// Check duration for each phase
positionExtrema := ruckig._profiles[0].Bound();
AssertEquals_LREAL(0.13645534129957551106, positionExtrema.Tmax, 1E-9, message:='Profile[0] Tmax incorrect');
AssertEquals_LREAL(-9.75706058924097519025, positionExtrema.Maximum, 1E-9, message:='Profile[0] maximum incorrect');
AssertEquals_LREAL(0.18561602058648316027, positionExtrema.Tmin, 1E-9, message:='Profile[0] Tmin incorrect');
AssertEquals_LREAL(-27.59745181479642894828, positionExtrema.Minimum, 1E-9, message:='Profile[0] minimum incorrect');

positionExtrema := ruckig._profiles[1].Bound();
AssertEquals_LREAL(0.18561602058648316027, positionExtrema.Tmax, 1E-9, message:='Profile[1] Tmax incorrect');
AssertEquals_LREAL(97.62295145618037395252, positionExtrema.Maximum, 1E-9, message:='Profile[1] maximum incorrect');
AssertEquals_LREAL(0.07177100934221260220, positionExtrema.Tmin, 1E-9, message:='Profile[1] Tmin incorrect');
AssertEquals_LREAL(33.68002966797480723926, positionExtrema.Minimum, 1E-9, message:='Profile[1] minimum incorrect');

positionExtrema := ruckig._profiles[2].Bound();
AssertEquals_LREAL(0.17125230195322679871, positionExtrema.Tmax, 1E-9, message:='Profile[2] Tmax incorrect');
AssertEquals_LREAL(-3.71520543795192104142, positionExtrema.Maximum, 1E-9, message:='Profile[2] maximum incorrect');
AssertEquals_LREAL(0.02823480242135182477, positionExtrema.Tmin, 1E-9, message:='Profile[2] Tmin incorrect');
AssertEquals_LREAL(-58.80508937654931855832, positionExtrema.Minimum, 1E-9, message:='Profile[2] minimum incorrect');
   

TEST_FINISHED();
END_METHOD

METHOD Test_Trajectory_HasTargetVelocity_17
VAR_INST
  ruckig : Struckig.Otg(0.001, 3) := (
  
    Synchronization := SynchronizationType.TimeSync,        
    MaxVelocity := [ 2000.00000000000000000000, 2000.00000000000000000000, 2000.00000000000000000000 ],
    MaxAcceleration := [ 20000.00000000000000000000, 20000.00000000000000000000, 20000.00000000000000000000 ],
    MaxJerk := [ 800000.00000000000000000000, 800000.00000000000000000000, 800000.00000000000000000000 ],
    CurrentPosition := [ 29.09201686409977583025, 26.79555889099025023370, -2.56405583533239678218 ],
    CurrentVelocity := [ -865.74515531652343725000, -446.66804096341445529106, 715.70430296883705523214 ],
    CurrentAcceleration := [ -419.53152796798531198874, 3725.90159379652868665289, 3083.71115629947962588631 ],
    TargetPosition := [ -5.98395477362167582669, 85.98880639059657937651, -77.56683653164213865239 ],
    TargetVelocity := [ -487.77111778150026566436, 597.93719815311010279402, -19.66112295679818089411 ],
    TargetAcceleration := [ 0.00000000000000000000, 0.00000000000000000000, 0.00000000000000000000 ]
  );
  
  positionExtrema : Struckig.ProfileBound;
END_VAR
TEST('Trajectory_HasTargetVelocity_17');

ruckig();

// Check total duration of profiles
AssertEquals_LREAL(Expected := 0.20727577661691312660, Actual := ruckig.Duration, DELTA := 1E-8, Message := 'Duration incorrect');

// Check duration for each phase
positionExtrema := ruckig._profiles[0].Bound();
AssertEquals_LREAL(0.00000000000000000000, positionExtrema.Tmax, 1E-9, message:='Profile[0] Tmax incorrect');
AssertEquals_LREAL(29.09201686409977583025, positionExtrema.Maximum, 1E-9, message:='Profile[0] maximum incorrect');
AssertEquals_LREAL(0.20727577661691309885, positionExtrema.Tmin, 1E-9, message:='Profile[0] Tmin incorrect');
AssertEquals_LREAL(-5.98395477362167582669, positionExtrema.Minimum, 1E-9, message:='Profile[0] minimum incorrect');

positionExtrema := ruckig._profiles[1].Bound();
AssertEquals_LREAL(0.20727577661691312660, positionExtrema.Tmax, 1E-9, message:='Profile[1] Tmax incorrect');
AssertEquals_LREAL(85.98880639059657937651, positionExtrema.Maximum, 1E-9, message:='Profile[1] maximum incorrect');
AssertEquals_LREAL(0.03742622748756373185, positionExtrema.Tmin, 1E-9, message:='Profile[1] Tmin incorrect');
AssertEquals_LREAL(19.01299187494276665689, positionExtrema.Minimum, 1E-9, message:='Profile[1] minimum incorrect');

positionExtrema := ruckig._profiles[2].Bound();
AssertEquals_LREAL(0.02885463894537435015, positionExtrema.Tmax, 1E-9, message:='Profile[2] Tmax incorrect');
AssertEquals_LREAL(16.16785534073141050726, positionExtrema.Maximum, 1E-9, message:='Profile[2] maximum incorrect');
AssertEquals_LREAL(0.20727577661691312660, positionExtrema.Tmin, 1E-9, message:='Profile[2] Tmin incorrect');
AssertEquals_LREAL(-77.56683653164213865239, positionExtrema.Minimum, 1E-9, message:='Profile[2] minimum incorrect');
   

TEST_FINISHED();
END_METHOD

METHOD Test_Trajectory_HasTargetVelocity_19
VAR_INST
  ruckig : Struckig.Otg(0.001, 3) := (
  
    Synchronization := SynchronizationType.TimeSync,        
    MaxVelocity := [ 2000.00000000000000000000, 2000.00000000000000000000, 2000.00000000000000000000 ],
    MaxAcceleration := [ 20000.00000000000000000000, 20000.00000000000000000000, 20000.00000000000000000000 ],
    MaxJerk := [ 800000.00000000000000000000, 800000.00000000000000000000, 800000.00000000000000000000 ],
    CurrentPosition := [ 80.71252725401120642346, 44.88025621959243949277, -12.15149697459605704353 ],
    CurrentVelocity := [ -948.15980924147334008012, -489.88340864146471176355, -827.37383618723242761916 ],
    CurrentAcceleration := [ -3514.54219608491530379979, -6906.59296787188577582128, 1315.32694212922615406569 ],
    TargetPosition := [ 59.95790772621657538366, -72.33902659712904892331, -15.83444921441858355138 ],
    TargetVelocity := [ -459.58488479420384464902, 187.24245841899073639070, 921.25657886294084164547 ],
    TargetAcceleration := [ 0.00000000000000000000, 0.00000000000000000000, 0.00000000000000000000 ]
  );
  
  positionExtrema : Struckig.ProfileBound;
END_VAR
TEST('Trajectory_HasTargetVelocity_19');

ruckig();

// Check total duration of profiles
AssertEquals_LREAL(Expected := 0.18063360611716061666, Actual := ruckig.Duration, DELTA := 1E-8, Message := 'Duration incorrect');

// Check duration for each phase
positionExtrema := ruckig._profiles[0].Bound();
AssertEquals_LREAL(0.00000000000000000000, positionExtrema.Tmax, 1E-9, message:='Profile[0] Tmax incorrect');
AssertEquals_LREAL(80.71252725401120642346, positionExtrema.Maximum, 1E-9, message:='Profile[0] maximum incorrect');
AssertEquals_LREAL(0.07992076514931607811, positionExtrema.Tmin, 1E-9, message:='Profile[0] Tmin incorrect');
AssertEquals_LREAL(44.57478735687137572086, positionExtrema.Minimum, 1E-9, message:='Profile[0] minimum incorrect');

positionExtrema := ruckig._profiles[1].Bound();
AssertEquals_LREAL(0.00000000000000000000, positionExtrema.Tmax, 1E-9, message:='Profile[1] Tmax incorrect');
AssertEquals_LREAL(44.88025621959243949277, positionExtrema.Maximum, 1E-9, message:='Profile[1] maximum incorrect');
AssertEquals_LREAL(0.15899784530207772271, positionExtrema.Tmin, 1E-9, message:='Profile[1] Tmin incorrect');
AssertEquals_LREAL(-75.03978196031663117083, positionExtrema.Minimum, 1E-9, message:='Profile[1] minimum incorrect');

positionExtrema := ruckig._profiles[2].Bound();
AssertEquals_LREAL(0.00000000000000000000, positionExtrema.Tmax, 1E-9, message:='Profile[2] Tmax incorrect');
AssertEquals_LREAL(-12.15149697459605704353, positionExtrema.Maximum, 1E-9, message:='Profile[2] maximum incorrect');
AssertEquals_LREAL(0.12139203206320470230, positionExtrema.Tmin, 1E-9, message:='Profile[2] Tmin incorrect');
AssertEquals_LREAL(-48.06891878044748267484, positionExtrema.Minimum, 1E-9, message:='Profile[2] minimum incorrect');
   

TEST_FINISHED();
END_METHOD

METHOD Test_Trajectory_HasTargetVelocity_20
VAR_INST
  ruckig : Struckig.Otg(0.001, 3) := (
  
    Synchronization := SynchronizationType.TimeSync,        
    MaxVelocity := [ 2000.00000000000000000000, 2000.00000000000000000000, 2000.00000000000000000000 ],
    MaxAcceleration := [ 20000.00000000000000000000, 20000.00000000000000000000, 20000.00000000000000000000 ],
    MaxJerk := [ 800000.00000000000000000000, 800000.00000000000000000000, 800000.00000000000000000000 ],
    CurrentPosition := [ 83.23209059023531608545, -91.01412900146218021291, -45.02313424428616883688 ],
    CurrentVelocity := [ 478.85135262944709211297, 941.48041828651457763044, 233.77464784894095828349 ],
    CurrentAcceleration := [ 4901.95944988452902180143, -711.94018044516997179016, -6268.14311607610761711840 ],
    TargetPosition := [ -60.31306848800090847362, -76.05388552166272120303, -77.88363097381802901964 ],
    TargetVelocity := [ -28.42585943091080480372, 112.61218905881105456501, -518.94659889602689872845 ],
    TargetAcceleration := [ 0.00000000000000000000, 0.00000000000000000000, 0.00000000000000000000 ]
  );
  
  positionExtrema : Struckig.ProfileBound;
END_VAR
TEST('Trajectory_HasTargetVelocity_20');

ruckig();

// Check total duration of profiles
AssertEquals_LREAL(Expected := 0.23417815197351798950, Actual := ruckig.Duration, DELTA := 1E-8, Message := 'Duration incorrect');

// Check duration for each phase
positionExtrema := ruckig._profiles[0].Bound();
AssertEquals_LREAL(0.03112744931235566018, positionExtrema.Tmax, 1E-9, message:='Profile[0] Tmax incorrect');
AssertEquals_LREAL(96.49098387500299622843, positionExtrema.Maximum, 1E-9, message:='Profile[0] maximum incorrect');
AssertEquals_LREAL(0.23417815197351798950, positionExtrema.Tmin, 1E-9, message:='Profile[0] Tmin incorrect');
AssertEquals_LREAL(-60.31306848800090847362, positionExtrema.Minimum, 1E-9, message:='Profile[0] minimum incorrect');

positionExtrema := ruckig._profiles[1].Bound();
AssertEquals_LREAL(0.05967434054652072384, positionExtrema.Tmax, 1E-9, message:='Profile[1] Tmax incorrect');
AssertEquals_LREAL(-58.39013538569540884282, positionExtrema.Maximum, 1E-9, message:='Profile[1] maximum incorrect');
AssertEquals_LREAL(0.00000000000000000000, positionExtrema.Tmin, 1E-9, message:='Profile[1] Tmin incorrect');
AssertEquals_LREAL(-91.01412900146218021291, positionExtrema.Minimum, 1E-9, message:='Profile[1] minimum incorrect');

positionExtrema := ruckig._profiles[2].Bound();
AssertEquals_LREAL(0.01824400060866057660, positionExtrema.Tmax, 1E-9, message:='Profile[2] Tmax incorrect');
AssertEquals_LREAL(-42.59202121085846926007, positionExtrema.Maximum, 1E-9, message:='Profile[2] maximum incorrect');
AssertEquals_LREAL(0.23417815197351793399, positionExtrema.Tmin, 1E-9, message:='Profile[2] Tmin incorrect');
AssertEquals_LREAL(-77.88363097381802901964, positionExtrema.Minimum, 1E-9, message:='Profile[2] minimum incorrect');
   

TEST_FINISHED();
END_METHOD

METHOD Test_Trajectory_HasTargetVelocity_21
VAR_INST
  ruckig : Struckig.Otg(0.001, 3) := (
  
    Synchronization := SynchronizationType.TimeSync,        
    MaxVelocity := [ 2000.00000000000000000000, 2000.00000000000000000000, 2000.00000000000000000000 ],
    MaxAcceleration := [ 20000.00000000000000000000, 20000.00000000000000000000, 20000.00000000000000000000 ],
    MaxJerk := [ 800000.00000000000000000000, 800000.00000000000000000000, 800000.00000000000000000000 ],
    CurrentPosition := [ -90.18105588355366819542, 11.40426253106177512109, -96.96426550769332664004 ],
    CurrentVelocity := [ 268.68366267133455949079, -230.39092451139003969729, 217.37624370386924965715 ],
    CurrentAcceleration := [ 6950.36478944877671892755, -1973.79956680386658263160, 9973.29839097329022479244 ],
    TargetPosition := [ 56.23264204687242795444, 89.78670651839811966965, 35.61941562712866016227 ],
    TargetVelocity := [ -748.79294734560005508683, 279.58550802373474652995, 329.97469268802092301485 ],
    TargetAcceleration := [ 0.00000000000000000000, 0.00000000000000000000, 0.00000000000000000000 ]
  );
  
  positionExtrema : Struckig.ProfileBound;
END_VAR
TEST('Trajectory_HasTargetVelocity_21');

ruckig();

// Check total duration of profiles
AssertEquals_LREAL(Expected := 0.22811513995984869507, Actual := ruckig.Duration, DELTA := 1E-8, Message := 'Duration incorrect');

// Check duration for each phase
positionExtrema := ruckig._profiles[0].Bound();
AssertEquals_LREAL(0.20311513995984870062, positionExtrema.Tmax, 1E-9, message:='Profile[0] Tmax incorrect');
AssertEquals_LREAL(72.86913239717907231352, positionExtrema.Maximum, 1E-9, message:='Profile[0] maximum incorrect');
AssertEquals_LREAL(0.00000000000000000000, positionExtrema.Tmin, 1E-9, message:='Profile[0] Tmin incorrect');
AssertEquals_LREAL(-90.18105588355366819542, positionExtrema.Minimum, 1E-9, message:='Profile[0] minimum incorrect');

positionExtrema := ruckig._profiles[1].Bound();
AssertEquals_LREAL(0.22811513995984869507, positionExtrema.Tmax, 1E-9, message:='Profile[1] Tmax incorrect');
AssertEquals_LREAL(89.78670651839811966965, positionExtrema.Maximum, 1E-9, message:='Profile[1] maximum incorrect');
AssertEquals_LREAL(0.02659326510902134191, positionExtrema.Tmin, 1E-9, message:='Profile[1] Tmin incorrect');
AssertEquals_LREAL(7.08705215721043568777, positionExtrema.Minimum, 1E-9, message:='Profile[1] minimum incorrect');

positionExtrema := ruckig._profiles[2].Bound();
AssertEquals_LREAL(0.22811513995984869507, positionExtrema.Tmax, 1E-9, message:='Profile[2] Tmax incorrect');
AssertEquals_LREAL(35.61941562712866016227, positionExtrema.Maximum, 1E-9, message:='Profile[2] maximum incorrect');
AssertEquals_LREAL(0.00000000000000000000, positionExtrema.Tmin, 1E-9, message:='Profile[2] Tmin incorrect');
AssertEquals_LREAL(-96.96426550769332664004, positionExtrema.Minimum, 1E-9, message:='Profile[2] minimum incorrect');
   

TEST_FINISHED();
END_METHOD

METHOD Test_Trajectory_HasTargetVelocity_22
VAR_INST
  ruckig : Struckig.Otg(0.001, 3) := (
  
    Synchronization := SynchronizationType.TimeSync,        
    MaxVelocity := [ 2000.00000000000000000000, 2000.00000000000000000000, 2000.00000000000000000000 ],
    MaxAcceleration := [ 20000.00000000000000000000, 20000.00000000000000000000, 20000.00000000000000000000 ],
    MaxJerk := [ 800000.00000000000000000000, 800000.00000000000000000000, 800000.00000000000000000000 ],
    CurrentPosition := [ -67.41063214653675572663, -34.84504669460216064181, 71.90844709145784463544 ],
    CurrentVelocity := [ -627.45307756820307076850, -697.56722522760969695810, -660.83791164052786371030 ],
    CurrentAcceleration := [ -7277.38846981411006709095, -2750.24172428648398636142, -978.85332476885741925798 ],
    TargetPosition := [ -57.66574268409263481772, -88.27667420321476754452, 96.97655926730644182499 ],
    TargetVelocity := [ -610.75498065854083051818, -654.20857948874163412256, 336.03100506981877515500 ],
    TargetAcceleration := [ 0.00000000000000000000, 0.00000000000000000000, 0.00000000000000000000 ]
  );
  
  positionExtrema : Struckig.ProfileBound;
END_VAR
TEST('Trajectory_HasTargetVelocity_22');

ruckig();

// Check total duration of profiles
AssertEquals_LREAL(Expected := 0.20245104517991782678, Actual := ruckig.Duration, DELTA := 1E-8, Message := 'Duration incorrect');

// Check duration for each phase
positionExtrema := ruckig._profiles[0].Bound();
AssertEquals_LREAL(0.17745104517991783233, positionExtrema.Tmax, 1E-9, message:='Profile[0] Tmax incorrect');
AssertEquals_LREAL(-44.48020150096243696680, positionExtrema.Maximum, 1E-9, message:='Profile[0] maximum incorrect');
AssertEquals_LREAL(0.03409673558726764031, positionExtrema.Tmin, 1E-9, message:='Profile[0] Tmin incorrect');
AssertEquals_LREAL(-87.74964255933160472978, positionExtrema.Minimum, 1E-9, message:='Profile[0] minimum incorrect');

positionExtrema := ruckig._profiles[1].Bound();
AssertEquals_LREAL(0.00000000000000000000, positionExtrema.Tmax, 1E-9, message:='Profile[1] Tmax incorrect');
AssertEquals_LREAL(-34.84504669460216064181, positionExtrema.Maximum, 1E-9, message:='Profile[1] maximum incorrect');
AssertEquals_LREAL(0.20245104517991779902, positionExtrema.Tmin, 1E-9, message:='Profile[1] Tmin incorrect');
AssertEquals_LREAL(-88.27667420321476754452, positionExtrema.Minimum, 1E-9, message:='Profile[1] minimum incorrect');

positionExtrema := ruckig._profiles[2].Bound();
AssertEquals_LREAL(0.20245104517991782678, positionExtrema.Tmax, 1E-9, message:='Profile[2] Tmax incorrect');
AssertEquals_LREAL(96.97655926730644182499, positionExtrema.Maximum, 1E-9, message:='Profile[2] maximum incorrect');
AssertEquals_LREAL(0.04944613992821229875, positionExtrema.Tmin, 1E-9, message:='Profile[2] Tmin incorrect');
AssertEquals_LREAL(52.48505260032155916861, positionExtrema.Minimum, 1E-9, message:='Profile[2] minimum incorrect');
   

TEST_FINISHED();
END_METHOD

METHOD Test_Trajectory_HasTargetVelocity_27
VAR_INST
  ruckig : Struckig.Otg(0.001, 3) := (
  
    Synchronization := SynchronizationType.TimeSync,        
    MaxVelocity := [ 2000.00000000000000000000, 2000.00000000000000000000, 2000.00000000000000000000 ],
    MaxAcceleration := [ 20000.00000000000000000000, 20000.00000000000000000000, 20000.00000000000000000000 ],
    MaxJerk := [ 800000.00000000000000000000, 800000.00000000000000000000, 800000.00000000000000000000 ],
    CurrentPosition := [ -29.47354331486815226526, 27.93495185982479256381, 25.04726746624395161689 ],
    CurrentVelocity := [ -230.41514646826715306815, -990.61050993041703804920, -730.89168845843755661917 ],
    CurrentAcceleration := [ 8742.55847153794820769690, 5915.09847409233043435961, 4511.30118221045631798916 ],
    TargetPosition := [ -46.00476070479609091990, -93.63874889974350423927, -84.98442462304464584122 ],
    TargetVelocity := [ 6.00636834947817987995, -353.84810777792165481515, -981.55918901141831156565 ],
    TargetAcceleration := [ 0.00000000000000000000, 0.00000000000000000000, 0.00000000000000000000 ]
  );
  
  positionExtrema : Struckig.ProfileBound;
END_VAR
TEST('Trajectory_HasTargetVelocity_27');

ruckig();

// Check total duration of profiles
AssertEquals_LREAL(Expected := 0.12586715797260131233, Actual := ruckig.Duration, DELTA := 1E-8, Message := 'Duration incorrect');

// Check duration for each phase
positionExtrema := ruckig._profiles[0].Bound();
AssertEquals_LREAL(0.00000000000000000000, positionExtrema.Tmax, 1E-9, message:='Profile[0] Tmax incorrect');
AssertEquals_LREAL(-29.47354331486815226526, positionExtrema.Maximum, 1E-9, message:='Profile[0] maximum incorrect');
AssertEquals_LREAL(0.12199211979553833962, positionExtrema.Tmin, 1E-9, message:='Profile[0] Tmin incorrect');
AssertEquals_LREAL(-46.02027730923590809198, positionExtrema.Minimum, 1E-9, message:='Profile[0] minimum incorrect');

positionExtrema := ruckig._profiles[1].Bound();
AssertEquals_LREAL(0.00000000000000000000, positionExtrema.Tmax, 1E-9, message:='Profile[1] Tmax incorrect');
AssertEquals_LREAL(27.93495185982479256381, positionExtrema.Maximum, 1E-9, message:='Profile[1] maximum incorrect');
AssertEquals_LREAL(0.12586715797260131233, positionExtrema.Tmin, 1E-9, message:='Profile[1] Tmin incorrect');
AssertEquals_LREAL(-93.63874889974350423927, positionExtrema.Minimum, 1E-9, message:='Profile[1] minimum incorrect');

positionExtrema := ruckig._profiles[2].Bound();
AssertEquals_LREAL(0.00000000000000000000, positionExtrema.Tmax, 1E-9, message:='Profile[2] Tmax incorrect');
AssertEquals_LREAL(25.04726746624395161689, positionExtrema.Maximum, 1E-9, message:='Profile[2] maximum incorrect');
AssertEquals_LREAL(0.12586715797260131233, positionExtrema.Tmin, 1E-9, message:='Profile[2] Tmin incorrect');
AssertEquals_LREAL(-84.98442462304464584122, positionExtrema.Minimum, 1E-9, message:='Profile[2] minimum incorrect');
   

TEST_FINISHED();
END_METHOD

METHOD Test_Trajectory_HasTargetVelocity_3
VAR_INST
  ruckig : Struckig.Otg(0.001, 3) := (
  
    Synchronization := SynchronizationType.TimeSync,        
    MaxVelocity := [ 2000.00000000000000000000, 2000.00000000000000000000, 2000.00000000000000000000 ],
    MaxAcceleration := [ 20000.00000000000000000000, 20000.00000000000000000000, 20000.00000000000000000000 ],
    MaxJerk := [ 800000.00000000000000000000, 800000.00000000000000000000, 800000.00000000000000000000 ],
    CurrentPosition := [ 26.53957997779905042535, -93.07095602825359037524, -22.16503543192527558858 ],
    CurrentVelocity := [ -978.47395774087203790259, 118.42434690487039006257, -240.97450183146906965703 ],
    CurrentAcceleration := [ 6077.24253675401814689394, 6138.16243012785889732186, -287.73427625073964009061 ],
    TargetPosition := [ -74.88074053142992170251, -34.02780494232007413302, 79.44667149152985530236 ],
    TargetVelocity := [ 90.05732775263027178880, 511.77846374302612275642, 384.28752753365688477061 ],
    TargetAcceleration := [ 0.00000000000000000000, 0.00000000000000000000, 0.00000000000000000000 ]
  );
  
  positionExtrema : Struckig.ProfileBound;
END_VAR
TEST('Trajectory_HasTargetVelocity_3');

ruckig();

// Check total duration of profiles
AssertEquals_LREAL(Expected := 0.16528629612631601242, Actual := ruckig.Duration, DELTA := 1E-8, Message := 'Duration incorrect');

// Check duration for each phase
positionExtrema := ruckig._profiles[0].Bound();
AssertEquals_LREAL(0.00000000000000000000, positionExtrema.Tmax, 1E-9, message:='Profile[0] Tmax incorrect');
AssertEquals_LREAL(26.53957997779905042535, positionExtrema.Maximum, 1E-9, message:='Profile[0] maximum incorrect');
AssertEquals_LREAL(0.15028151957411181594, positionExtrema.Tmin, 1E-9, message:='Profile[0] Tmin incorrect');
AssertEquals_LREAL(-75.78160058464112580623, positionExtrema.Minimum, 1E-9, message:='Profile[0] minimum incorrect');

positionExtrema := ruckig._profiles[1].Bound();
AssertEquals_LREAL(0.16528629612631601242, positionExtrema.Tmax, 1E-9, message:='Profile[1] Tmax incorrect');
AssertEquals_LREAL(-34.02780494232007413302, positionExtrema.Maximum, 1E-9, message:='Profile[1] maximum incorrect');
AssertEquals_LREAL(0.00000000000000000000, positionExtrema.Tmin, 1E-9, message:='Profile[1] Tmin incorrect');
AssertEquals_LREAL(-93.07095602825359037524, positionExtrema.Minimum, 1E-9, message:='Profile[1] minimum incorrect');

positionExtrema := ruckig._profiles[2].Bound();
AssertEquals_LREAL(0.16528629612631601242, positionExtrema.Tmax, 1E-9, message:='Profile[2] Tmax incorrect');
AssertEquals_LREAL(79.44667149152985530236, positionExtrema.Maximum, 1E-9, message:='Profile[2] maximum incorrect');
AssertEquals_LREAL(0.02490687981607753870, positionExtrema.Tmin, 1E-9, message:='Profile[2] Tmin incorrect');
AssertEquals_LREAL(-26.19606685654071753788, positionExtrema.Minimum, 1E-9, message:='Profile[2] minimum incorrect');
   

TEST_FINISHED();
END_METHOD

METHOD Test_Trajectory_HasTargetVelocity_34
VAR_INST
  ruckig : Struckig.Otg(0.001, 3) := (
  
    Synchronization := SynchronizationType.TimeSync,        
    MaxVelocity := [ 2000.00000000000000000000, 2000.00000000000000000000, 2000.00000000000000000000 ],
    MaxAcceleration := [ 20000.00000000000000000000, 20000.00000000000000000000, 20000.00000000000000000000 ],
    MaxJerk := [ 800000.00000000000000000000, 800000.00000000000000000000, 800000.00000000000000000000 ],
    CurrentPosition := [ 52.72619781679460970736, -25.78201897219773286452, 80.53760009793651875043 ],
    CurrentVelocity := [ -120.69783207836667315860, 178.50171370384009605914, -265.96277737557261389156 ],
    CurrentAcceleration := [ 9869.62339068779328954406, 8236.73224664633380598389, 4587.35631399299018085003 ],
    TargetPosition := [ -7.31302355801524583967, 98.53124939615054245223, -70.22704739896117587250 ],
    TargetVelocity := [ 648.92680228108224582684, 640.55767309494626715605, -28.66025813343185291160 ],
    TargetAcceleration := [ 0.00000000000000000000, 0.00000000000000000000, 0.00000000000000000000 ]
  );
  
  positionExtrema : Struckig.ProfileBound;
END_VAR
TEST('Trajectory_HasTargetVelocity_34');

ruckig();

// Check total duration of profiles
AssertEquals_LREAL(Expected := 0.19340758597333415625, Actual := ruckig.Duration, DELTA := 1E-8, Message := 'Duration incorrect');

// Check duration for each phase
positionExtrema := ruckig._profiles[0].Bound();
AssertEquals_LREAL(0.00000000000000000000, positionExtrema.Tmax, 1E-9, message:='Profile[0] Tmax incorrect');
AssertEquals_LREAL(52.72619781679460970736, positionExtrema.Maximum, 1E-9, message:='Profile[0] maximum incorrect');
AssertEquals_LREAL(0.16840758597333416180, positionExtrema.Tmin, 1E-9, message:='Profile[0] Tmin incorrect');
AssertEquals_LREAL(-21.45286028170894354616, positionExtrema.Minimum, 1E-9, message:='Profile[0] minimum incorrect');

positionExtrema := ruckig._profiles[1].Bound();
AssertEquals_LREAL(0.19340758597333415625, positionExtrema.Tmax, 1E-9, message:='Profile[1] Tmax incorrect');
AssertEquals_LREAL(98.53124939615054245223, positionExtrema.Maximum, 1E-9, message:='Profile[1] maximum incorrect');
AssertEquals_LREAL(0.00000000000000000000, positionExtrema.Tmin, 1E-9, message:='Profile[1] Tmin incorrect');
AssertEquals_LREAL(-25.78201897219773286452, positionExtrema.Minimum, 1E-9, message:='Profile[1] minimum incorrect');

positionExtrema := ruckig._profiles[2].Bound();
AssertEquals_LREAL(0.00000000000000000000, positionExtrema.Tmax, 1E-9, message:='Profile[2] Tmax incorrect');
AssertEquals_LREAL(80.53760009793651875043, positionExtrema.Maximum, 1E-9, message:='Profile[2] maximum incorrect');
AssertEquals_LREAL(0.19340758597333415625, positionExtrema.Tmin, 1E-9, message:='Profile[2] Tmin incorrect');
AssertEquals_LREAL(-70.22704739896117587250, positionExtrema.Minimum, 1E-9, message:='Profile[2] minimum incorrect');
   

TEST_FINISHED();
END_METHOD

METHOD Test_Trajectory_HasTargetVelocity_35
VAR_INST
  ruckig : Struckig.Otg(0.001, 3) := (
  
    Synchronization := SynchronizationType.TimeSync,        
    MaxVelocity := [ 2000.00000000000000000000, 2000.00000000000000000000, 2000.00000000000000000000 ],
    MaxAcceleration := [ 20000.00000000000000000000, 20000.00000000000000000000, 20000.00000000000000000000 ],
    MaxJerk := [ 800000.00000000000000000000, 800000.00000000000000000000, 800000.00000000000000000000 ],
    CurrentPosition := [ -34.17551015513085133080, -36.11913195800440234962, 51.20006403327516864010 ],
    CurrentVelocity := [ -436.11356880285654824547, -175.40667275745920505869, 746.11367552095180144534 ],
    CurrentAcceleration := [ -9866.78282408208724518772, -2137.40956356850620068144, 2870.77810427219810662791 ],
    TargetPosition := [ 94.89098874895094581916, -43.87608688101931875281, 99.33475834942979076914 ],
    TargetVelocity := [ 945.80038372223793885496, -169.18944510068342879094, 349.24092684862353053177 ],
    TargetAcceleration := [ 0.00000000000000000000, 0.00000000000000000000, 0.00000000000000000000 ]
  );
  
  positionExtrema : Struckig.ProfileBound;
END_VAR
TEST('Trajectory_HasTargetVelocity_35');

ruckig();

// Check total duration of profiles
AssertEquals_LREAL(Expected := 0.19433376507479860340, Actual := ruckig.Duration, DELTA := 1E-8, Message := 'Duration incorrect');

// Check duration for each phase
positionExtrema := ruckig._profiles[0].Bound();
AssertEquals_LREAL(0.19433376507479860340, positionExtrema.Tmax, 1E-9, message:='Profile[0] Tmax incorrect');
AssertEquals_LREAL(94.89098874895094581916, positionExtrema.Maximum, 1E-9, message:='Profile[0] maximum incorrect');
AssertEquals_LREAL(0.03733347853010261091, positionExtrema.Tmin, 1E-9, message:='Profile[0] Tmin incorrect');
AssertEquals_LREAL(-50.39525451816182055609, positionExtrema.Minimum, 1E-9, message:='Profile[0] minimum incorrect');

positionExtrema := ruckig._profiles[1].Bound();
AssertEquals_LREAL(0.00000000000000000000, positionExtrema.Tmax, 1E-9, message:='Profile[1] Tmax incorrect');
AssertEquals_LREAL(-36.11913195800440234962, positionExtrema.Maximum, 1E-9, message:='Profile[1] maximum incorrect');
AssertEquals_LREAL(0.19433376507479860340, positionExtrema.Tmin, 1E-9, message:='Profile[1] Tmin incorrect');
AssertEquals_LREAL(-43.87608688101931875281, positionExtrema.Minimum, 1E-9, message:='Profile[1] minimum incorrect');

positionExtrema := ruckig._profiles[2].Bound();
AssertEquals_LREAL(0.19433376507479860340, positionExtrema.Tmax, 1E-9, message:='Profile[2] Tmax incorrect');
AssertEquals_LREAL(99.33475834942979076914, positionExtrema.Maximum, 1E-9, message:='Profile[2] maximum incorrect');
AssertEquals_LREAL(0.00000000000000000000, positionExtrema.Tmin, 1E-9, message:='Profile[2] Tmin incorrect');
AssertEquals_LREAL(51.20006403327516864010, positionExtrema.Minimum, 1E-9, message:='Profile[2] minimum incorrect');
   

TEST_FINISHED();
END_METHOD

METHOD Test_Trajectory_HasTargetVelocity_36
VAR_INST
  ruckig : Struckig.Otg(0.001, 3) := (
  
    Synchronization := SynchronizationType.TimeSync,        
    MaxVelocity := [ 2000.00000000000000000000, 2000.00000000000000000000, 2000.00000000000000000000 ],
    MaxAcceleration := [ 20000.00000000000000000000, 20000.00000000000000000000, 20000.00000000000000000000 ],
    MaxJerk := [ 800000.00000000000000000000, 800000.00000000000000000000, 800000.00000000000000000000 ],
    CurrentPosition := [ 64.35804589046725254775, -17.92542582379405757820, 1.48297994216896711350 ],
    CurrentVelocity := [ 464.92943892208950273925, -779.25597761349285974575, 998.42982599227457285451 ],
    CurrentAcceleration := [ 4749.41918638301285682246, -6355.94416374630964128301, 521.38908747176901670173 ],
    TargetPosition := [ 90.33897695077399703223, -51.53109090258827507114, -18.12118447758692241223 ],
    TargetVelocity := [ 651.93427968717173826008, 22.75188801650608638738, 576.72189974234174769663 ],
    TargetAcceleration := [ 0.00000000000000000000, 0.00000000000000000000, 0.00000000000000000000 ]
  );
  
  positionExtrema : Struckig.ProfileBound;
END_VAR
TEST('Trajectory_HasTargetVelocity_36');

ruckig();

// Check total duration of profiles
AssertEquals_LREAL(Expected := 0.22796271730102146691, Actual := ruckig.Duration, DELTA := 1E-8, Message := 'Duration incorrect');

// Check duration for each phase
positionExtrema := ruckig._profiles[0].Bound();
AssertEquals_LREAL(0.22796271730102146691, positionExtrema.Tmax, 1E-9, message:='Profile[0] Tmax incorrect');
AssertEquals_LREAL(90.33897695077399703223, positionExtrema.Maximum, 1E-9, message:='Profile[0] maximum incorrect');
AssertEquals_LREAL(0.00000000000000000000, positionExtrema.Tmin, 1E-9, message:='Profile[0] Tmin incorrect');
AssertEquals_LREAL(64.35804589046725254775, positionExtrema.Minimum, 1E-9, message:='Profile[0] minimum incorrect');

positionExtrema := ruckig._profiles[1].Bound();
AssertEquals_LREAL(0.00000000000000000000, positionExtrema.Tmax, 1E-9, message:='Profile[1] Tmax incorrect');
AssertEquals_LREAL(-17.92542582379405757820, positionExtrema.Maximum, 1E-9, message:='Profile[1] maximum incorrect');
AssertEquals_LREAL(0.21997970156554483290, positionExtrema.Tmin, 1E-9, message:='Profile[1] Tmin incorrect');
AssertEquals_LREAL(-51.64657663770686468752, positionExtrema.Minimum, 1E-9, message:='Profile[1] minimum incorrect');

positionExtrema := ruckig._profiles[2].Bound();
AssertEquals_LREAL(0.09985417258924977890, positionExtrema.Tmax, 1E-9, message:='Profile[2] Tmax incorrect');
AssertEquals_LREAL(25.50333501341721742506, positionExtrema.Maximum, 1E-9, message:='Profile[2] maximum incorrect');
AssertEquals_LREAL(0.20296271730102147246, positionExtrema.Tmin, 1E-9, message:='Profile[2] Tmin incorrect');
AssertEquals_LREAL(-30.45589863781214745586, positionExtrema.Minimum, 1E-9, message:='Profile[2] minimum incorrect');
   

TEST_FINISHED();
END_METHOD

METHOD Test_Trajectory_HasTargetVelocity_4
VAR_INST
  ruckig : Struckig.Otg(0.001, 3) := (
  
    Synchronization := SynchronizationType.TimeSync,        
    MaxVelocity := [ 2000.00000000000000000000, 2000.00000000000000000000, 2000.00000000000000000000 ],
    MaxAcceleration := [ 20000.00000000000000000000, 20000.00000000000000000000, 20000.00000000000000000000 ],
    MaxJerk := [ 800000.00000000000000000000, 800000.00000000000000000000, 800000.00000000000000000000 ],
    CurrentPosition := [ 39.65544040447574047903, -16.66018211442579399773, -58.50720512248746274508 ],
    CurrentVelocity := [ 152.61039713388095151458, -842.85004717237586646661, -233.59739104574180146301 ],
    CurrentAcceleration := [ -6325.89065787396975792944, -1505.68574067445842956658, -3102.88067432900697895093 ],
    TargetPosition := [ -66.91581266696782392955, -93.61689817230509902402, 29.78308499537988041084 ],
    TargetVelocity := [ 439.82482428242337846314, -284.79407434788117825519, -482.50326392108468098741 ],
    TargetAcceleration := [ 0.00000000000000000000, 0.00000000000000000000, 0.00000000000000000000 ]
  );
  
  positionExtrema : Struckig.ProfileBound;
END_VAR
TEST('Trajectory_HasTargetVelocity_4');

ruckig();

// Check total duration of profiles
AssertEquals_LREAL(Expected := 0.21237444505671645989, Actual := ruckig.Duration, DELTA := 1E-8, Message := 'Duration incorrect');

// Check duration for each phase
positionExtrema := ruckig._profiles[0].Bound();
AssertEquals_LREAL(0.01316518724815633583, positionExtrema.Tmax, 1E-9, message:='Profile[0] Tmax incorrect');
AssertEquals_LREAL(40.81213387351741772591, positionExtrema.Maximum, 1E-9, message:='Profile[0] maximum incorrect');
AssertEquals_LREAL(0.18737444505671646544, positionExtrema.Tmin, 1E-9, message:='Profile[0] Tmin incorrect');
AssertEquals_LREAL(-75.82809994069509684778, positionExtrema.Minimum, 1E-9, message:='Profile[0] minimum incorrect');

positionExtrema := ruckig._profiles[1].Bound();
AssertEquals_LREAL(0.00000000000000000000, positionExtrema.Tmax, 1E-9, message:='Profile[1] Tmax incorrect');
AssertEquals_LREAL(-16.66018211442579399773, positionExtrema.Maximum, 1E-9, message:='Profile[1] maximum incorrect');
AssertEquals_LREAL(0.21237444505671648765, positionExtrema.Tmin, 1E-9, message:='Profile[1] Tmin incorrect');
AssertEquals_LREAL(-93.61689817230509902402, positionExtrema.Minimum, 1E-9, message:='Profile[1] minimum incorrect');

positionExtrema := ruckig._profiles[2].Bound();
AssertEquals_LREAL(0.18737444505671646544, positionExtrema.Tmax, 1E-9, message:='Profile[2] Tmax incorrect');
AssertEquals_LREAL(39.76233326007365320720, positionExtrema.Maximum, 1E-9, message:='Profile[2] maximum incorrect');
AssertEquals_LREAL(0.02835383367352977552, positionExtrema.Tmin, 1E-9, message:='Profile[2] Tmin incorrect');
AssertEquals_LREAL(-63.33854775889894028751, positionExtrema.Minimum, 1E-9, message:='Profile[2] minimum incorrect');
   

TEST_FINISHED();
END_METHOD

METHOD Test_Trajectory_HasTargetVelocity_44
VAR_INST
  ruckig : Struckig.Otg(0.001, 3) := (
  
    Synchronization := SynchronizationType.TimeSync,        
    MaxVelocity := [ 2000.00000000000000000000, 2000.00000000000000000000, 2000.00000000000000000000 ],
    MaxAcceleration := [ 20000.00000000000000000000, 20000.00000000000000000000, 20000.00000000000000000000 ],
    MaxJerk := [ 800000.00000000000000000000, 800000.00000000000000000000, 800000.00000000000000000000 ],
    CurrentPosition := [ 33.20927605983496277986, 90.97207853642058239529, -55.08094735406923092569 ],
    CurrentVelocity := [ -992.30424733188726804656, -901.32445813848187299300, 586.66877088523051497759 ],
    CurrentAcceleration := [ -2055.28947681546742387582, -6947.94625488244855660014, 5257.19066749439298291691 ],
    TargetPosition := [ 67.40661968603291143154, 85.00720295179675645159, 88.22002633481628208756 ],
    TargetVelocity := [ -402.53524157043091236119, -775.84245093694903516734, -256.32808117758236221562 ],
    TargetAcceleration := [ 0.00000000000000000000, 0.00000000000000000000, 0.00000000000000000000 ]
  );
  
  positionExtrema : Struckig.ProfileBound;
END_VAR
TEST('Trajectory_HasTargetVelocity_44');

ruckig();

// Check total duration of profiles
AssertEquals_LREAL(Expected := 0.23151950260302325835, Actual := ruckig.Duration, DELTA := 1E-8, Message := 'Duration incorrect');

// Check duration for each phase
positionExtrema := ruckig._profiles[0].Bound();
AssertEquals_LREAL(0.20651950260302323614, positionExtrema.Tmax, 1E-9, message:='Profile[0] Tmax incorrect');
AssertEquals_LREAL(75.38666739196018795610, positionExtrema.Maximum, 1E-9, message:='Profile[0] maximum incorrect');
AssertEquals_LREAL(0.10082888716067818502, positionExtrema.Tmin, 1E-9, message:='Profile[0] Tmin incorrect');
AssertEquals_LREAL(6.96062616300369274569, positionExtrema.Minimum, 1E-9, message:='Profile[0] minimum incorrect');

positionExtrema := ruckig._profiles[1].Bound();
AssertEquals_LREAL(0.20651950260302326390, positionExtrema.Tmax, 1E-9, message:='Profile[1] Tmax incorrect');
AssertEquals_LREAL(102.31993089188715373439, positionExtrema.Maximum, 1E-9, message:='Profile[1] maximum incorrect');
AssertEquals_LREAL(0.09899354847148797432, positionExtrema.Tmin, 1E-9, message:='Profile[1] Tmin incorrect');
AssertEquals_LREAL(59.91000069944395534094, positionExtrema.Minimum, 1E-9, message:='Profile[1] minimum incorrect');

positionExtrema := ruckig._profiles[2].Bound();
AssertEquals_LREAL(0.20651950260302326390, positionExtrema.Tmax, 1E-9, message:='Profile[2] Tmax incorrect');
AssertEquals_LREAL(92.54489503092254665262, positionExtrema.Maximum, 1E-9, message:='Profile[2] maximum incorrect');
AssertEquals_LREAL(0.00000000000000000000, positionExtrema.Tmin, 1E-9, message:='Profile[2] Tmin incorrect');
AssertEquals_LREAL(-55.08094735406923092569, positionExtrema.Minimum, 1E-9, message:='Profile[2] minimum incorrect');
   

TEST_FINISHED();
END_METHOD

METHOD Test_Trajectory_HasTargetVelocity_45
VAR_INST
  ruckig : Struckig.Otg(0.001, 3) := (
  
    Synchronization := SynchronizationType.TimeSync,        
    MaxVelocity := [ 2000.00000000000000000000, 2000.00000000000000000000, 2000.00000000000000000000 ],
    MaxAcceleration := [ 20000.00000000000000000000, 20000.00000000000000000000, 20000.00000000000000000000 ],
    MaxJerk := [ 800000.00000000000000000000, 800000.00000000000000000000, 800000.00000000000000000000 ],
    CurrentPosition := [ 94.90826698124541849211, 98.68601680143464704997, -94.06931326171563512162 ],
    CurrentVelocity := [ -430.89473663668559311191, -312.79662986488631304383, -992.83444762482452006225 ],
    CurrentAcceleration := [ -5676.65368720607239083620, -3762.56637347724063147325, 6550.62068049420850002207 ],
    TargetPosition := [ -39.76061431821072034154, -54.28480859989317508507, 99.44666750072161676144 ],
    TargetVelocity := [ -859.34940974039534467011, 795.33260348280805374088, -780.22698676244044690975 ],
    TargetAcceleration := [ 0.00000000000000000000, 0.00000000000000000000, 0.00000000000000000000 ]
  );
  
  positionExtrema : Struckig.ProfileBound;
END_VAR
TEST('Trajectory_HasTargetVelocity_45');

ruckig();

// Check total duration of profiles
AssertEquals_LREAL(Expected := 0.33133845625565350179, Actual := ruckig.Duration, DELTA := 1E-8, Message := 'Duration incorrect');

// Check duration for each phase
positionExtrema := ruckig._profiles[0].Bound();
AssertEquals_LREAL(0.00000000000000000000, positionExtrema.Tmax, 1E-9, message:='Profile[0] Tmax incorrect');
AssertEquals_LREAL(94.90826698124541849211, positionExtrema.Maximum, 1E-9, message:='Profile[0] maximum incorrect');
AssertEquals_LREAL(0.33133845625565355730, positionExtrema.Tmin, 1E-9, message:='Profile[0] Tmin incorrect');
AssertEquals_LREAL(-39.76061431821072034154, positionExtrema.Minimum, 1E-9, message:='Profile[0] minimum incorrect');

positionExtrema := ruckig._profiles[1].Bound();
AssertEquals_LREAL(0.00000000000000000000, positionExtrema.Tmax, 1E-9, message:='Profile[1] Tmax incorrect');
AssertEquals_LREAL(98.68601680143464704997, positionExtrema.Maximum, 1E-9, message:='Profile[1] maximum incorrect');
AssertEquals_LREAL(0.25596921475835221482, positionExtrema.Tmin, 1E-9, message:='Profile[1] Tmin incorrect');
AssertEquals_LREAL(-74.18217506467304644957, positionExtrema.Minimum, 1E-9, message:='Profile[1] minimum incorrect');

positionExtrema := ruckig._profiles[2].Bound();
AssertEquals_LREAL(0.30633845625565347959, positionExtrema.Tmax, 1E-9, message:='Profile[2] Tmax incorrect');
AssertEquals_LREAL(116.86900883644932491734, positionExtrema.Maximum, 1E-9, message:='Profile[2] maximum incorrect');
AssertEquals_LREAL(0.01681172414938223933, positionExtrema.Tmin, 1E-9, message:='Profile[2] Tmin incorrect');
AssertEquals_LREAL(-109.20131569941064242357, positionExtrema.Minimum, 1E-9, message:='Profile[2] minimum incorrect');
   

TEST_FINISHED();
END_METHOD

METHOD Test_Trajectory_HasTargetVelocity_54
VAR_INST
  ruckig : Struckig.Otg(0.001, 3) := (
  
    Synchronization := SynchronizationType.TimeSync,        
    MaxVelocity := [ 2000.00000000000000000000, 2000.00000000000000000000, 2000.00000000000000000000 ],
    MaxAcceleration := [ 20000.00000000000000000000, 20000.00000000000000000000, 20000.00000000000000000000 ],
    MaxJerk := [ 800000.00000000000000000000, 800000.00000000000000000000, 800000.00000000000000000000 ],
    CurrentPosition := [ 97.11911830820099567063, -34.96974423375549179127, -12.00449667266771314189 ],
    CurrentVelocity := [ 732.45673588056706648786, -364.10592093846560146631, 417.20885103824889483803 ],
    CurrentAcceleration := [ -7499.05473487195013149176, -3391.82282403053886810085, -1045.80444633833030820824 ],
    TargetPosition := [ -34.58240005713176401514, -14.14677543732022968470, -36.27520430827089370496 ],
    TargetVelocity := [ -912.82558763807946888846, 208.36586640296604855394, -568.50539307151495904691 ],
    TargetAcceleration := [ 0.00000000000000000000, 0.00000000000000000000, 0.00000000000000000000 ]
  );
  
  positionExtrema : Struckig.ProfileBound;
END_VAR
TEST('Trajectory_HasTargetVelocity_54');

ruckig();

// Check total duration of profiles
AssertEquals_LREAL(Expected := 0.18808008069304424370, Actual := ruckig.Duration, DELTA := 1E-8, Message := 'Duration incorrect');

// Check duration for each phase
positionExtrema := ruckig._profiles[0].Bound();
AssertEquals_LREAL(0.01562618158141006186, positionExtrema.Tmax, 1E-9, message:='Profile[0] Tmax incorrect');
AssertEquals_LREAL(107.14032815468360126943, positionExtrema.Maximum, 1E-9, message:='Profile[0] maximum incorrect');
AssertEquals_LREAL(0.18808008069304424370, positionExtrema.Tmin, 1E-9, message:='Profile[0] Tmin incorrect');
AssertEquals_LREAL(-34.58240005713176401514, positionExtrema.Minimum, 1E-9, message:='Profile[0] minimum incorrect');

positionExtrema := ruckig._profiles[1].Bound();
AssertEquals_LREAL(0.18808008069304424370, positionExtrema.Tmax, 1E-9, message:='Profile[1] Tmax incorrect');
AssertEquals_LREAL(-14.14677543732022968470, positionExtrema.Maximum, 1E-9, message:='Profile[1] maximum incorrect');
AssertEquals_LREAL(0.03540881837579783198, positionExtrema.Tmin, 1E-9, message:='Profile[1] Tmin incorrect');
AssertEquals_LREAL(-44.10216499913330778782, positionExtrema.Minimum, 1E-9, message:='Profile[1] minimum incorrect');

positionExtrema := ruckig._profiles[2].Bound();
AssertEquals_LREAL(0.03261360243271873433, positionExtrema.Tmax, 1E-9, message:='Profile[2] Tmax incorrect');
AssertEquals_LREAL(-3.46659095127397254288, positionExtrema.Maximum, 1E-9, message:='Profile[2] maximum incorrect');
AssertEquals_LREAL(0.18808008069304424370, positionExtrema.Tmin, 1E-9, message:='Profile[2] Tmin incorrect');
AssertEquals_LREAL(-36.27520430827089370496, positionExtrema.Minimum, 1E-9, message:='Profile[2] minimum incorrect');
   

TEST_FINISHED();
END_METHOD

METHOD Test_Trajectory_HasTargetVelocity_55
VAR_INST
  ruckig : Struckig.Otg(0.001, 3) := (
  
    Synchronization := SynchronizationType.TimeSync,        
    MaxVelocity := [ 2000.00000000000000000000, 2000.00000000000000000000, 2000.00000000000000000000 ],
    MaxAcceleration := [ 20000.00000000000000000000, 20000.00000000000000000000, 20000.00000000000000000000 ],
    MaxJerk := [ 800000.00000000000000000000, 800000.00000000000000000000, 800000.00000000000000000000 ],
    CurrentPosition := [ 93.14320777040134657909, -89.74312540741888710727, -99.44513086937998025405 ],
    CurrentVelocity := [ 358.10280009786106347747, 608.03888639331830745505, 352.36242097628496594552 ],
    CurrentAcceleration := [ 2330.07739343047796864994, 9276.80286875897945719771, 5318.79396039618404756766 ],
    TargetPosition := [ 90.69471017690091230179, -41.60077247517397580623, 88.58596356723177223103 ],
    TargetVelocity := [ -791.02326773343907007074, -519.34342102358630199888, -658.93165900614667407353 ],
    TargetAcceleration := [ 0.00000000000000000000, 0.00000000000000000000, 0.00000000000000000000 ]
  );
  
  positionExtrema : Struckig.ProfileBound;
END_VAR
TEST('Trajectory_HasTargetVelocity_55');

ruckig();

// Check total duration of profiles
AssertEquals_LREAL(Expected := 0.24005299536906613000, Actual := ruckig.Duration, DELTA := 1E-8, Message := 'Duration incorrect');

// Check duration for each phase
positionExtrema := ruckig._profiles[0].Bound();
AssertEquals_LREAL(0.18612405983992955094, positionExtrema.Tmax, 1E-9, message:='Profile[0] Tmax incorrect');
AssertEquals_LREAL(115.79065190073221458533, positionExtrema.Maximum, 1E-9, message:='Profile[0] maximum incorrect');
AssertEquals_LREAL(0.24005299536906613000, positionExtrema.Tmin, 1E-9, message:='Profile[0] Tmin incorrect');
AssertEquals_LREAL(90.69471017690091230179, positionExtrema.Minimum, 1E-9, message:='Profile[0] minimum incorrect');

positionExtrema := ruckig._profiles[1].Bound();
AssertEquals_LREAL(0.20158118915996722786, positionExtrema.Tmax, 1E-9, message:='Profile[1] Tmax incorrect');
AssertEquals_LREAL(-28.88685866039741512168, positionExtrema.Maximum, 1E-9, message:='Profile[1] maximum incorrect');
AssertEquals_LREAL(0.00000000000000000000, positionExtrema.Tmin, 1E-9, message:='Profile[1] Tmin incorrect');
AssertEquals_LREAL(-89.74312540741888710727, positionExtrema.Minimum, 1E-9, message:='Profile[1] minimum incorrect');

positionExtrema := ruckig._profiles[2].Bound();
AssertEquals_LREAL(0.21505299536906613556, positionExtrema.Tmax, 1E-9, message:='Profile[2] Tmax incorrect');
AssertEquals_LREAL(102.97592170905214459253, positionExtrema.Maximum, 1E-9, message:='Profile[2] maximum incorrect');
AssertEquals_LREAL(0.00000000000000000000, positionExtrema.Tmin, 1E-9, message:='Profile[2] Tmin incorrect');
AssertEquals_LREAL(-99.44513086937998025405, positionExtrema.Minimum, 1E-9, message:='Profile[2] minimum incorrect');
   

TEST_FINISHED();
END_METHOD

METHOD Test_Trajectory_HasTargetVelocity_69
VAR_INST
  ruckig : Struckig.Otg(0.001, 3) := (
  
    Synchronization := SynchronizationType.TimeSync,        
    MaxVelocity := [ 2000.00000000000000000000, 2000.00000000000000000000, 2000.00000000000000000000 ],
    MaxAcceleration := [ 20000.00000000000000000000, 20000.00000000000000000000, 20000.00000000000000000000 ],
    MaxJerk := [ 800000.00000000000000000000, 800000.00000000000000000000, 800000.00000000000000000000 ],
    CurrentPosition := [ 57.27064181935406850243, 60.77262566521827125143, 62.27255646349433959585 ],
    CurrentVelocity := [ 537.97467176664963517396, -420.66138587481805188872, -215.06636530667026363517 ],
    CurrentAcceleration := [ -1444.96134368556158733554, -9785.35194497229167609476, -7380.59859225371474167332 ],
    TargetPosition := [ -63.84344825014372304395, -56.97669545923665168630, -22.85605311820776819332 ],
    TargetVelocity := [ -201.51935759086109101190, 630.98179272467473310826, 276.24214614430115943833 ],
    TargetAcceleration := [ 0.00000000000000000000, 0.00000000000000000000, 0.00000000000000000000 ]
  );
  
  positionExtrema : Struckig.ProfileBound;
END_VAR
TEST('Trajectory_HasTargetVelocity_69');

ruckig();

// Check total duration of profiles
AssertEquals_LREAL(Expected := 0.20486873141224784534, Actual := ruckig.Duration, DELTA := 1E-8, Message := 'Duration incorrect');

// Check duration for each phase
positionExtrema := ruckig._profiles[0].Bound();
AssertEquals_LREAL(0.02319379832039304701, positionExtrema.Tmax, 1E-9, message:='Profile[0] Tmax incorrect');
AssertEquals_LREAL(67.69603683932946580626, positionExtrema.Maximum, 1E-9, message:='Profile[0] maximum incorrect');
AssertEquals_LREAL(0.20486873141224784534, positionExtrema.Tmin, 1E-9, message:='Profile[0] Tmin incorrect');
AssertEquals_LREAL(-63.84344825014372304395, positionExtrema.Minimum, 1E-9, message:='Profile[0] minimum incorrect');

positionExtrema := ruckig._profiles[1].Bound();
AssertEquals_LREAL(0.00000000000000000000, positionExtrema.Tmax, 1E-9, message:='Profile[1] Tmax incorrect');
AssertEquals_LREAL(60.77262566521827125143, positionExtrema.Maximum, 1E-9, message:='Profile[1] maximum incorrect');
AssertEquals_LREAL(0.17986873141224785089, positionExtrema.Tmin, 1E-9, message:='Profile[1] Tmin incorrect');
AssertEquals_LREAL(-70.66790694402018857545, positionExtrema.Minimum, 1E-9, message:='Profile[1] minimum incorrect');

positionExtrema := ruckig._profiles[2].Bound();
AssertEquals_LREAL(0.00000000000000000000, positionExtrema.Tmax, 1E-9, message:='Profile[2] Tmax incorrect');
AssertEquals_LREAL(62.27255646349433959585, positionExtrema.Maximum, 1E-9, message:='Profile[2] maximum incorrect');
AssertEquals_LREAL(0.17986873141224782313, positionExtrema.Tmin, 1E-9, message:='Profile[2] Tmin incorrect');
AssertEquals_LREAL(-27.67877343848196147746, positionExtrema.Minimum, 1E-9, message:='Profile[2] minimum incorrect');
   

TEST_FINISHED();
END_METHOD

METHOD Test_Trajectory_HasTargetVelocity_9
VAR_INST
  ruckig : Struckig.Otg(0.001, 3) := (
  
    Synchronization := SynchronizationType.TimeSync,        
    MaxVelocity := [ 2000.00000000000000000000, 2000.00000000000000000000, 2000.00000000000000000000 ],
    MaxAcceleration := [ 20000.00000000000000000000, 20000.00000000000000000000, 20000.00000000000000000000 ],
    MaxJerk := [ 800000.00000000000000000000, 800000.00000000000000000000, 800000.00000000000000000000 ],
    CurrentPosition := [ 51.69848597185645644458, 7.44342383280722685868, 34.92442688172334896990 ],
    CurrentVelocity := [ -421.44916669967597044888, -275.10229321522490408825, 914.94627896365750530094 ],
    CurrentAcceleration := [ 8837.53563716822463902645, -8661.28092822574944875669, -64.93681698721775319427 ],
    TargetPosition := [ 85.87288052559532047781, -50.28620894086743930984, -15.14712281129145310388 ],
    TargetVelocity := [ 635.15347000890233175596, 546.48145876800276710128, 277.88896365954042266821 ],
    TargetAcceleration := [ 0.00000000000000000000, 0.00000000000000000000, 0.00000000000000000000 ]
  );
  
  positionExtrema : Struckig.ProfileBound;
END_VAR
TEST('Trajectory_HasTargetVelocity_9');

ruckig();

// Check total duration of profiles
AssertEquals_LREAL(Expected := 0.21938772367288389420, Actual := ruckig.Duration, DELTA := 1E-8, Message := 'Duration incorrect');

// Check duration for each phase
positionExtrema := ruckig._profiles[0].Bound();
AssertEquals_LREAL(0.21938772367288389420, positionExtrema.Tmax, 1E-9, message:='Profile[0] Tmax incorrect');
AssertEquals_LREAL(85.87288052559532047781, positionExtrema.Maximum, 1E-9, message:='Profile[0] maximum incorrect');
AssertEquals_LREAL(0.02559956417752039248, positionExtrema.Tmin, 1E-9, message:='Profile[0] Tmin incorrect');
AssertEquals_LREAL(45.80781253564739330386, positionExtrema.Minimum, 1E-9, message:='Profile[0] minimum incorrect');

positionExtrema := ruckig._profiles[1].Bound();
AssertEquals_LREAL(0.00000000000000000000, positionExtrema.Tmax, 1E-9, message:='Profile[1] Tmax incorrect');
AssertEquals_LREAL(7.44342383280722685868, positionExtrema.Maximum, 1E-9, message:='Profile[1] maximum incorrect');
AssertEquals_LREAL(0.17034751041817919326, positionExtrema.Tmin, 1E-9, message:='Profile[1] Tmin incorrect');
AssertEquals_LREAL(-63.21307103826610074293, positionExtrema.Minimum, 1E-9, message:='Profile[1] minimum incorrect');

positionExtrema := ruckig._profiles[2].Bound();
AssertEquals_LREAL(0.02491882897876597849, positionExtrema.Tmax, 1E-9, message:='Profile[2] Tmax incorrect');
AssertEquals_LREAL(55.64054914337343404895, positionExtrema.Maximum, 1E-9, message:='Profile[2] maximum incorrect');
AssertEquals_LREAL(0.19438772367288389975, positionExtrema.Tmin, 1E-9, message:='Profile[2] Tmin incorrect');
AssertEquals_LREAL(-20.01101356944660381032, positionExtrema.Minimum, 1E-9, message:='Profile[2] minimum incorrect');
   

TEST_FINISHED();
END_METHOD

END_FUNCTION_BLOCK

// ---- POUs/TargetPosVelAccTest.TcPOU
FUNCTION_BLOCK TargetPosVelAccTest EXTENDS TcUnit_Zeugwerk.FB_TestSuite
VAR
  ruckig : Struckig.Otg(0.001, 3) := (
  
    Synchronization := SynchronizationType.TimeSync,        
    MaxVelocity := [ 2000.00000000000000000000, 2000.00000000000000000000, 2000.00000000000000000000 ],
    MaxAcceleration := [ 20000.00000000000000000000, 20000.00000000000000000000, 20000.00000000000000000000 ],
    MaxJerk := [ 800000.00000000000000000000, 800000.00000000000000000000, 800000.00000000000000000000 ],
    CurrentPosition := [ 48.86656216713086564596, 31.55963588984187140341, -13.09422790776093847853 ],
    CurrentVelocity := [ -274.21841080128081102885, -440.94461360926254656079, -764.75678162210920163488 ],
    CurrentAcceleration := [ -1478.09700836416959646158, 686.79611869591644790489, -9263.72976579731221136171 ],
    TargetPosition := [ 25.57994474955607699940, -15.83091418217283319336, -38.97164514571973370494 ],
    TargetVelocity := [ 0.00000000000000000000, 0.00000000000000000000, 0.00000000000000000000 ],
    TargetAcceleration := [ 0.00000000000000000000, 0.00000000000000000000, 0.00000000000000000000 ]
  );
  
  positionExtrema : Struckig.ProfileBound;  
END_VAR

Test_Trajectory_HasTargetVelocity_HasTargetAcceleration_10();
Test_Trajectory_HasTargetVelocity_HasTargetAcceleration_11();
Test_Trajectory_HasTargetVelocity_HasTargetAcceleration_13();
Test_Trajectory_HasTargetVelocity_HasTargetAcceleration_23();
Test_Trajectory_HasTargetVelocity_HasTargetAcceleration_24();
Test_Trajectory_HasTargetVelocity_HasTargetAcceleration_25();
Test_Trajectory_HasTargetVelocity_HasTargetAcceleration_28();
Test_Trajectory_HasTargetVelocity_HasTargetAcceleration_31();
Test_Trajectory_HasTargetVelocity_HasTargetAcceleration_38();
Test_Trajectory_HasTargetVelocity_HasTargetAcceleration_41();
Test_Trajectory_HasTargetVelocity_HasTargetAcceleration_46();
Test_Trajectory_HasTargetVelocity_HasTargetAcceleration_47();
Test_Trajectory_HasTargetVelocity_HasTargetAcceleration_48();
Test_Trajectory_HasTargetVelocity_HasTargetAcceleration_51();
Test_Trajectory_HasTargetVelocity_HasTargetAcceleration_56();
Test_Trajectory_HasTargetVelocity_HasTargetAcceleration_60();
Test_Trajectory_HasTargetVelocity_HasTargetAcceleration_61();
Test_Trajectory_HasTargetVelocity_HasTargetAcceleration_66();
Test_Trajectory_HasTargetVelocity_HasTargetAcceleration_70();

METHOD Test_Trajectory_HasTargetVelocity_HasTargetAcceleration_10
VAR_INST
  ruckig : Struckig.Otg(0.001, 3) := (
  
    Synchronization := SynchronizationType.TimeSync,        
    MaxVelocity := [ 2000.00000000000000000000, 2000.00000000000000000000, 2000.00000000000000000000 ],
    MaxAcceleration := [ 20000.00000000000000000000, 20000.00000000000000000000, 20000.00000000000000000000 ],
    MaxJerk := [ 800000.00000000000000000000, 800000.00000000000000000000, 800000.00000000000000000000 ],
    CurrentPosition := [ -39.47806403569489219763, 85.51350241283674336046, 44.68502449548182653416 ],
    CurrentVelocity := [ 850.44438005471602082253, -488.80559496892584547822, -700.94733690949385618296 ],
    CurrentAcceleration := [ -1858.32224098730875994079, -3187.99589590553750895197, 92.02409562680077215191 ],
    TargetPosition := [ 62.43779038863485197908, 75.32481099920960332383, 88.50314116872792169488 ],
    TargetVelocity := [ 123.28060327403977680660, 99.93105645665400516009, -988.17694465354713884153 ],
    TargetAcceleration := [ 523.22114524957532921690, -244.33148184356286947150, -78.54730785107437895931 ]
  );
  
  positionExtrema : Struckig.ProfileBound;
END_VAR
TEST('Trajectory_HasTargetVelocity_HasTargetAcceleration_10');

ruckig();

// Check total duration of profiles
AssertEquals_LREAL(Expected := 0.25386401433668925876, Actual := ruckig.Duration, DELTA := 1E-8, Message := 'Duration incorrect');

// Check duration for each phase
positionExtrema := ruckig._profiles[0].Bound();
AssertEquals_LREAL(0.25386401433668925876, positionExtrema.Tmax, 1E-9, message:='Profile[0] Tmax incorrect');
AssertEquals_LREAL(62.43779038863485197908, positionExtrema.Maximum, 1E-9, message:='Profile[0] maximum incorrect');
AssertEquals_LREAL(0.00000000000000000000, positionExtrema.Tmin, 1E-9, message:='Profile[0] Tmin incorrect');
AssertEquals_LREAL(-39.47806403569489219763, positionExtrema.Minimum, 1E-9, message:='Profile[0] minimum incorrect');

positionExtrema := ruckig._profiles[1].Bound();
AssertEquals_LREAL(0.00000000000000000000, positionExtrema.Tmax, 1E-9, message:='Profile[1] Tmax incorrect');
AssertEquals_LREAL(85.51350241283674336046, positionExtrema.Maximum, 1E-9, message:='Profile[1] maximum incorrect');
AssertEquals_LREAL(0.04836149122526862271, positionExtrema.Tmin, 1E-9, message:='Profile[1] Tmin incorrect');
AssertEquals_LREAL(71.36198278424123486730, positionExtrema.Minimum, 1E-9, message:='Profile[1] minimum incorrect');

positionExtrema := ruckig._profiles[2].Bound();
AssertEquals_LREAL(0.22896219847150309223, positionExtrema.Tmax, 1E-9, message:='Profile[2] Tmax incorrect');
AssertEquals_LREAL(111.02730430222078439328, positionExtrema.Maximum, 1E-9, message:='Profile[2] maximum incorrect');
AssertEquals_LREAL(0.02488496988046649816, positionExtrema.Tmin, 1E-9, message:='Profile[2] Tmin incorrect');
AssertEquals_LREAL(29.32517254863061850756, positionExtrema.Minimum, 1E-9, message:='Profile[2] minimum incorrect');
   

TEST_FINISHED();
END_METHOD

METHOD Test_Trajectory_HasTargetVelocity_HasTargetAcceleration_11
VAR_INST
  ruckig : Struckig.Otg(0.001, 3) := (
  
    Synchronization := SynchronizationType.TimeSync,        
    MaxVelocity := [ 2000.00000000000000000000, 2000.00000000000000000000, 2000.00000000000000000000 ],
    MaxAcceleration := [ 20000.00000000000000000000, 20000.00000000000000000000, 20000.00000000000000000000 ],
    MaxJerk := [ 800000.00000000000000000000, 800000.00000000000000000000, 800000.00000000000000000000 ],
    CurrentPosition := [ -11.00969981377717488158, 79.30083386555023139408, -79.33289322247576080827 ],
    CurrentVelocity := [ 340.34781182329970761202, 246.68864182540505680663, -994.15213442746357941360 ],
    CurrentAcceleration := [ 8700.39687173053971491754, -5148.82815689879680576269, 8397.80808154643818852492 ],
    TargetPosition := [ 10.69516269239538530655, -19.77457066315008660240, -45.65505563877125894123 ],
    TargetVelocity := [ -427.08539049490741490445, -334.25491167273139581084, -671.08698082447017441154 ],
    TargetAcceleration := [ 932.74239593593802055693, -718.28804857432260178030, 358.92850741837651185051 ]
  );
  
  positionExtrema : Struckig.ProfileBound;
END_VAR
TEST('Trajectory_HasTargetVelocity_HasTargetAcceleration_11');

ruckig();

// Check total duration of profiles
AssertEquals_LREAL(Expected := 0.23152173952640786592, Actual := ruckig.Duration, DELTA := 1E-8, Message := 'Duration incorrect');

// Check duration for each phase
positionExtrema := ruckig._profiles[0].Bound();
AssertEquals_LREAL(0.19546951360492895167, positionExtrema.Tmax, 1E-9, message:='Profile[0] Tmax incorrect');
AssertEquals_LREAL(20.62712040740557739582, positionExtrema.Maximum, 1E-9, message:='Profile[0] maximum incorrect');
AssertEquals_LREAL(0.00000000000000000000, positionExtrema.Tmin, 1E-9, message:='Profile[0] Tmin incorrect');
AssertEquals_LREAL(-11.00969981377717488158, positionExtrema.Minimum, 1E-9, message:='Profile[0] minimum incorrect');

positionExtrema := ruckig._profiles[1].Bound();
AssertEquals_LREAL(0.01856396480387650233, positionExtrema.Tmax, 1E-9, message:='Profile[1] Tmax incorrect');
AssertEquals_LREAL(82.14015275808480964770, positionExtrema.Maximum, 1E-9, message:='Profile[1] maximum incorrect');
AssertEquals_LREAL(0.23152173952640786592, positionExtrema.Tmin, 1E-9, message:='Profile[1] Tmin incorrect');
AssertEquals_LREAL(-19.77457066315008660240, positionExtrema.Minimum, 1E-9, message:='Profile[1] minimum incorrect');

positionExtrema := ruckig._profiles[2].Bound();
AssertEquals_LREAL(0.20607307889213488661, positionExtrema.Tmax, 1E-9, message:='Profile[2] Tmax incorrect');
AssertEquals_LREAL(-30.65808709370843132547, positionExtrema.Maximum, 1E-9, message:='Profile[2] maximum incorrect');
AssertEquals_LREAL(0.01450273989806695300, positionExtrema.Tmin, 1E-9, message:='Profile[2] Tmin incorrect');
AssertEquals_LREAL(-92.46095600628422062073, positionExtrema.Minimum, 1E-9, message:='Profile[2] minimum incorrect');
   

TEST_FINISHED();
END_METHOD

METHOD Test_Trajectory_HasTargetVelocity_HasTargetAcceleration_13
VAR_INST
  ruckig : Struckig.Otg(0.001, 3) := (
  
    Synchronization := SynchronizationType.TimeSync,        
    MaxVelocity := [ 2000.00000000000000000000, 2000.00000000000000000000, 2000.00000000000000000000 ],
    MaxAcceleration := [ 20000.00000000000000000000, 20000.00000000000000000000, 20000.00000000000000000000 ],
    MaxJerk := [ 800000.00000000000000000000, 800000.00000000000000000000, 800000.00000000000000000000 ],
    CurrentPosition := [ 9.69881262256657805665, 49.09528145802553922294, 90.83813935322746146994 ],
    CurrentVelocity := [ -433.54343331398354166595, 472.80041396309707124601, 363.83131582274700122070 ],
    CurrentAcceleration := [ 4083.49957317767075437587, 8321.57042699825615272857, 3041.72021404646875453182 ],
    TargetPosition := [ -40.75433231777056874989, 5.53885291167379989474, 72.17019091605928338140 ],
    TargetVelocity := [ 43.64296519726190126676, -988.37442788621763156698, 453.07334546629840588139 ],
    TargetAcceleration := [ 36.30955223704063428158, 458.49955170826592620870, 185.69577899128807985107 ]
  );
  
  positionExtrema : Struckig.ProfileBound;
END_VAR
TEST('Trajectory_HasTargetVelocity_HasTargetAcceleration_13');

ruckig();

// Check total duration of profiles
AssertEquals_LREAL(Expected := 0.16126678162936489147, Actual := ruckig.Duration, DELTA := 1E-8, Message := 'Duration incorrect');

// Check duration for each phase
positionExtrema := ruckig._profiles[0].Bound();
AssertEquals_LREAL(0.00000000000000000000, positionExtrema.Tmax, 1E-9, message:='Profile[0] Tmax incorrect');
AssertEquals_LREAL(9.69881262256657805665, positionExtrema.Maximum, 1E-9, message:='Profile[0] maximum incorrect');
AssertEquals_LREAL(0.15086662057218858113, positionExtrema.Tmin, 1E-9, message:='Profile[0] Tmin incorrect');
AssertEquals_LREAL(-41.05627366867881988810, positionExtrema.Minimum, 1E-9, message:='Profile[0] minimum incorrect');

positionExtrema := ruckig._profiles[1].Bound();
AssertEquals_LREAL(0.06070813242930364617, positionExtrema.Tmax, 1E-9, message:='Profile[1] Tmax incorrect');
AssertEquals_LREAL(65.46161526012338072178, positionExtrema.Maximum, 1E-9, message:='Profile[1] maximum incorrect');
AssertEquals_LREAL(0.16126678162936489147, positionExtrema.Tmin, 1E-9, message:='Profile[1] Tmin incorrect');
AssertEquals_LREAL(5.53885291167379989474, positionExtrema.Minimum, 1E-9, message:='Profile[1] minimum incorrect');

positionExtrema := ruckig._profiles[2].Bound();
AssertEquals_LREAL(0.02880215026755808538, positionExtrema.Tmax, 1E-9, message:='Profile[2] Tmax incorrect');
AssertEquals_LREAL(99.39315110411790499256, positionExtrema.Maximum, 1E-9, message:='Profile[2] maximum incorrect');
AssertEquals_LREAL(0.13649890135310399630, positionExtrema.Tmin, 1E-9, message:='Profile[2] Tmin incorrect');
AssertEquals_LREAL(63.03132241192619744652, positionExtrema.Minimum, 1E-9, message:='Profile[2] minimum incorrect');
   

TEST_FINISHED();
END_METHOD

METHOD Test_Trajectory_HasTargetVelocity_HasTargetAcceleration_23
VAR_INST
  ruckig : Struckig.Otg(0.001, 3) := (
  
    Synchronization := SynchronizationType.TimeSync,        
    MaxVelocity := [ 2000.00000000000000000000, 2000.00000000000000000000, 2000.00000000000000000000 ],
    MaxAcceleration := [ 20000.00000000000000000000, 20000.00000000000000000000, 20000.00000000000000000000 ],
    MaxJerk := [ 800000.00000000000000000000, 800000.00000000000000000000, 800000.00000000000000000000 ],
    CurrentPosition := [ 47.53700980033448786344, -67.27694012280542779081, -86.38486619516218922854 ],
    CurrentVelocity := [ 624.06318776028729189420, -26.67222535829409935104, 867.31073468942531690118 ],
    CurrentAcceleration := [ 8661.05253784820160944946, 1127.19399458656334900297, -862.51135134606010979041 ],
    TargetPosition := [ -44.06957139861784611412, -0.35301738432740137341, 34.14509493445279986190 ],
    TargetVelocity := [ -953.23022651827614026843, -141.30450499696496535762, 399.93502902002660448488 ],
    TargetAcceleration := [ -153.89029587917991648283, 786.51386102503238362260, -59.28726062308271593793 ]
  );
  
  positionExtrema : Struckig.ProfileBound;
END_VAR
TEST('Trajectory_HasTargetVelocity_HasTargetAcceleration_23');

ruckig();

// Check total duration of profiles
AssertEquals_LREAL(Expected := 0.18439257781618231813, Actual := ruckig.Duration, DELTA := 1E-8, Message := 'Duration incorrect');

// Check duration for each phase
positionExtrema := ruckig._profiles[0].Bound();
AssertEquals_LREAL(0.03582631567231025355, positionExtrema.Tmax, 1E-9, message:='Profile[0] Tmax incorrect');
AssertEquals_LREAL(69.32203709773510524883, positionExtrema.Maximum, 1E-9, message:='Profile[0] maximum incorrect');
AssertEquals_LREAL(0.18439257781618231813, positionExtrema.Tmin, 1E-9, message:='Profile[0] Tmin incorrect');
AssertEquals_LREAL(-44.06957139861784611412, positionExtrema.Minimum, 1E-9, message:='Profile[0] minimum incorrect');

positionExtrema := ruckig._profiles[1].Bound();
AssertEquals_LREAL(0.16458849419234267142, positionExtrema.Tmax, 1E-9, message:='Profile[1] Tmax incorrect');
AssertEquals_LREAL(1.56399878718463591909, positionExtrema.Maximum, 1E-9, message:='Profile[1] maximum incorrect');
AssertEquals_LREAL(0.00687749187842422172, positionExtrema.Tmin, 1E-9, message:='Profile[1] Tmin incorrect');
AssertEquals_LREAL(-67.39034610548161197130, positionExtrema.Minimum, 1E-9, message:='Profile[1] minimum incorrect');

positionExtrema := ruckig._profiles[2].Bound();
AssertEquals_LREAL(0.18439257781618231813, positionExtrema.Tmax, 1E-9, message:='Profile[2] Tmax incorrect');
AssertEquals_LREAL(34.14509493445279986190, positionExtrema.Maximum, 1E-9, message:='Profile[2] maximum incorrect');
AssertEquals_LREAL(0.00000000000000000000, positionExtrema.Tmin, 1E-9, message:='Profile[2] Tmin incorrect');
AssertEquals_LREAL(-86.38486619516218922854, positionExtrema.Minimum, 1E-9, message:='Profile[2] minimum incorrect');
   

TEST_FINISHED();
END_METHOD

METHOD Test_Trajectory_HasTargetVelocity_HasTargetAcceleration_24
VAR_INST
  ruckig : Struckig.Otg(0.001, 3) := (
  
    Synchronization := SynchronizationType.TimeSync,        
    MaxVelocity := [ 2000.00000000000000000000, 2000.00000000000000000000, 2000.00000000000000000000 ],
    MaxAcceleration := [ 20000.00000000000000000000, 20000.00000000000000000000, 20000.00000000000000000000 ],
    MaxJerk := [ 800000.00000000000000000000, 800000.00000000000000000000, 800000.00000000000000000000 ],
    CurrentPosition := [ 55.38049842099269426399, -36.51718980157055227664, 46.34633267231370723493 ],
    CurrentVelocity := [ -275.90586981683884459926, 325.28418297116309076955, -569.40991459537576702132 ],
    CurrentAcceleration := [ -4904.07330886993440799415, 6037.59143415146354527678, 285.12822918885831313673 ],
    TargetPosition := [ 35.43064875422174964115, 95.51797326506493845955, 58.54459913513463220625 ],
    TargetVelocity := [ 257.68447580225415549648, 639.68339605466303510184, -872.58228531132567695749 ],
    TargetAcceleration := [ -374.50768793212057516939, 123.04281317134154960513, 26.25305058742901564983 ]
  );
  
  positionExtrema : Struckig.ProfileBound;
END_VAR
TEST('Trajectory_HasTargetVelocity_HasTargetAcceleration_24');

ruckig();

// Check total duration of profiles
AssertEquals_LREAL(Expected := 0.20661176225146463126, Actual := ruckig.Duration, DELTA := 1E-8, Message := 'Duration incorrect');

// Check duration for each phase
positionExtrema := ruckig._profiles[0].Bound();
AssertEquals_LREAL(0.00000000000000000000, positionExtrema.Tmax, 1E-9, message:='Profile[0] Tmax incorrect');
AssertEquals_LREAL(55.38049842099269426399, positionExtrema.Maximum, 1E-9, message:='Profile[0] maximum incorrect');
AssertEquals_LREAL(0.18000578842985828776, positionExtrema.Tmin, 1E-9, message:='Profile[0] Tmin incorrect');
AssertEquals_LREAL(30.93057238685970133929, positionExtrema.Minimum, 1E-9, message:='Profile[0] minimum incorrect');

positionExtrema := ruckig._profiles[1].Bound();
AssertEquals_LREAL(0.20661176225146460350, positionExtrema.Tmax, 1E-9, message:='Profile[1] Tmax incorrect');
AssertEquals_LREAL(95.51797326506493845955, positionExtrema.Maximum, 1E-9, message:='Profile[1] maximum incorrect');
AssertEquals_LREAL(0.00000000000000000000, positionExtrema.Tmin, 1E-9, message:='Profile[1] Tmin incorrect');
AssertEquals_LREAL(-36.51718980157055227664, positionExtrema.Minimum, 1E-9, message:='Profile[1] minimum incorrect');

positionExtrema := ruckig._profiles[2].Bound();
AssertEquals_LREAL(0.12053321807179237513, positionExtrema.Tmax, 1E-9, message:='Profile[2] Tmax incorrect');
AssertEquals_LREAL(79.04467479917035177550, positionExtrema.Maximum, 1E-9, message:='Profile[2] maximum incorrect');
AssertEquals_LREAL(0.02464358971351392896, positionExtrema.Tmin, 1E-9, message:='Profile[2] Tmin incorrect');
AssertEquals_LREAL(34.39610348174581133662, positionExtrema.Minimum, 1E-9, message:='Profile[2] minimum incorrect');
   

TEST_FINISHED();
END_METHOD

METHOD Test_Trajectory_HasTargetVelocity_HasTargetAcceleration_25
VAR_INST
  ruckig : Struckig.Otg(0.001, 3) := (
  
    Synchronization := SynchronizationType.TimeSync,        
    MaxVelocity := [ 2000.00000000000000000000, 2000.00000000000000000000, 2000.00000000000000000000 ],
    MaxAcceleration := [ 20000.00000000000000000000, 20000.00000000000000000000, 20000.00000000000000000000 ],
    MaxJerk := [ 800000.00000000000000000000, 800000.00000000000000000000, 800000.00000000000000000000 ],
    CurrentPosition := [ -43.61348212315061800837, 29.83034818219718431465, 49.28274589774380842755 ],
    CurrentVelocity := [ 445.78248483783545452752, -365.97477149155758979759, 834.21346728548428473005 ],
    CurrentAcceleration := [ 8151.27766250318381935358, 4550.14049799841450294480, -5778.56226010059071995784 ],
    TargetPosition := [ -60.34727868985516607836, -0.54575471898803584736, -65.76232312596496853985 ],
    TargetVelocity := [ 256.22760642234447914234, -829.37836652808050530439, -911.71719060686370994517 ],
    TargetAcceleration := [ 190.44282430417842988390, 16.22894859941652612179, -320.27777449957079625165 ]
  );
  
  positionExtrema : Struckig.ProfileBound;
END_VAR
TEST('Trajectory_HasTargetVelocity_HasTargetAcceleration_25');

ruckig();

// Check total duration of profiles
AssertEquals_LREAL(Expected := 0.18857033031718306582, Actual := ruckig.Duration, DELTA := 1E-8, Message := 'Duration incorrect');

// Check duration for each phase
positionExtrema := ruckig._profiles[0].Bound();
AssertEquals_LREAL(0.05441964492405890197, positionExtrema.Tmax, 1E-9, message:='Profile[0] Tmax incorrect');
AssertEquals_LREAL(-27.82441980071925158313, positionExtrema.Maximum, 1E-9, message:='Profile[0] maximum incorrect');
AssertEquals_LREAL(0.16380838384756329917, positionExtrema.Tmin, 1E-9, message:='Profile[0] Tmin incorrect');
AssertEquals_LREAL(-64.60920272819178933332, positionExtrema.Minimum, 1E-9, message:='Profile[0] minimum incorrect');

positionExtrema := ruckig._profiles[1].Bound();
AssertEquals_LREAL(0.00000000000000000000, positionExtrema.Tmax, 1E-9, message:='Profile[1] Tmax incorrect');
AssertEquals_LREAL(29.83034818219718431465, positionExtrema.Maximum, 1E-9, message:='Profile[1] maximum incorrect');
AssertEquals_LREAL(0.18857033031718306582, positionExtrema.Tmin, 1E-9, message:='Profile[1] Tmin incorrect');
AssertEquals_LREAL(-0.54575471898803584736, positionExtrema.Minimum, 1E-9, message:='Profile[1] minimum incorrect');

positionExtrema := ruckig._profiles[2].Bound();
AssertEquals_LREAL(0.01777679717487426134, positionExtrema.Tmax, 1E-9, message:='Profile[2] Tmax incorrect');
AssertEquals_LREAL(62.45030459150993351614, positionExtrema.Maximum, 1E-9, message:='Profile[2] maximum incorrect');
AssertEquals_LREAL(0.18857033031718306582, positionExtrema.Tmin, 1E-9, message:='Profile[2] Tmin incorrect');
AssertEquals_LREAL(-65.76232312596496853985, positionExtrema.Minimum, 1E-9, message:='Profile[2] minimum incorrect');
   

TEST_FINISHED();
END_METHOD

METHOD Test_Trajectory_HasTargetVelocity_HasTargetAcceleration_28
VAR_INST
  ruckig : Struckig.Otg(0.001, 3) := (
  
    Synchronization := SynchronizationType.TimeSync,        
    MaxVelocity := [ 2000.00000000000000000000, 2000.00000000000000000000, 2000.00000000000000000000 ],
    MaxAcceleration := [ 20000.00000000000000000000, 20000.00000000000000000000, 20000.00000000000000000000 ],
    MaxJerk := [ 800000.00000000000000000000, 800000.00000000000000000000, 800000.00000000000000000000 ],
    CurrentPosition := [ -25.75950331902309642373, 25.28257521119543582699, 29.01217051002615221478 ],
    CurrentVelocity := [ -258.16394237742667883140, 916.64967525581641893950, -53.97433058993919985369 ],
    CurrentAcceleration := [ -9538.00892060086152923759, 3140.62431203669075330254, 714.16116385760506091174 ],
    TargetPosition := [ -99.15720752840965701580, -11.85176568807662533800, -0.99133804973871519906 ],
    TargetVelocity := [ -12.33203202805157161492, -43.09141691856916622783, 791.12283404668596631382 ],
    TargetAcceleration := [ -865.12500750031517782190, 291.33729215361222486536, -357.67243570276048103551 ]
  );
  
  positionExtrema : Struckig.ProfileBound;
END_VAR
TEST('Trajectory_HasTargetVelocity_HasTargetAcceleration_28');

ruckig();

// Check total duration of profiles
AssertEquals_LREAL(Expected := 0.19601934217339064825, Actual := ruckig.Duration, DELTA := 1E-8, Message := 'Duration incorrect');

// Check duration for each phase
positionExtrema := ruckig._profiles[0].Bound();
AssertEquals_LREAL(0.00000000000000000000, positionExtrema.Tmax, 1E-9, message:='Profile[0] Tmax incorrect');
AssertEquals_LREAL(-25.75950331902309642373, positionExtrema.Maximum, 1E-9, message:='Profile[0] maximum incorrect');
AssertEquals_LREAL(0.19601934217339067601, positionExtrema.Tmin, 1E-9, message:='Profile[0] Tmin incorrect');
AssertEquals_LREAL(-99.15720752840965701580, positionExtrema.Minimum, 1E-9, message:='Profile[0] minimum incorrect');

positionExtrema := ruckig._profiles[1].Bound();
AssertEquals_LREAL(0.02892578039004586529, positionExtrema.Tmax, 1E-9, message:='Profile[1] Tmax incorrect');
AssertEquals_LREAL(49.88430076962359294157, positionExtrema.Maximum, 1E-9, message:='Profile[1] maximum incorrect');
AssertEquals_LREAL(0.19601934217339064825, positionExtrema.Tmin, 1E-9, message:='Profile[1] Tmin incorrect');
AssertEquals_LREAL(-11.85176568807662533800, positionExtrema.Minimum, 1E-9, message:='Profile[1] minimum incorrect');

positionExtrema := ruckig._profiles[2].Bound();
AssertEquals_LREAL(0.00000000000000000000, positionExtrema.Tmax, 1E-9, message:='Profile[2] Tmax incorrect');
AssertEquals_LREAL(29.01217051002615221478, positionExtrema.Maximum, 1E-9, message:='Profile[2] maximum incorrect');
AssertEquals_LREAL(0.13019418227345949668, positionExtrema.Tmin, 1E-9, message:='Profile[2] Tmin incorrect');
AssertEquals_LREAL(-24.59064078002127473610, positionExtrema.Minimum, 1E-9, message:='Profile[2] minimum incorrect');
   

TEST_FINISHED();
END_METHOD

METHOD Test_Trajectory_HasTargetVelocity_HasTargetAcceleration_31
VAR_INST
  ruckig : Struckig.Otg(0.001, 3) := (
  
    Synchronization := SynchronizationType.TimeSync,        
    MaxVelocity := [ 2000.00000000000000000000, 2000.00000000000000000000, 2000.00000000000000000000 ],
    MaxAcceleration := [ 20000.00000000000000000000, 20000.00000000000000000000, 20000.00000000000000000000 ],
    MaxJerk := [ 800000.00000000000000000000, 800000.00000000000000000000, 800000.00000000000000000000 ],
    CurrentPosition := [ -54.94342725690739825950, -71.16344937395382430623, -99.92141940871530891854 ],
    CurrentVelocity := [ 203.04708462957614756306, -87.88615914847480325989, -244.40742200449426491105 ],
    CurrentAcceleration := [ -9414.24830241836389177479, 3433.58972946014000626747, -1048.10905719350193976425 ],
    TargetPosition := [ -30.34627507739200780179, 41.33313071646210801191, 94.47974487226861128875 ],
    TargetVelocity := [ -104.33706621689987059654, -659.36109838358197521302, 811.33117925934993763804 ],
    TargetAcceleration := [ 523.43053514200096287823, 100.75104632855459385610, 320.80199262854853259341 ]
  );
  
  positionExtrema : Struckig.ProfileBound;
END_VAR
TEST('Trajectory_HasTargetVelocity_HasTargetAcceleration_31');

ruckig();

// Check total duration of profiles
AssertEquals_LREAL(Expected := 0.22338925049474450679, Actual := ruckig.Duration, DELTA := 1E-8, Message := 'Duration incorrect');

// Check duration for each phase
positionExtrema := ruckig._profiles[0].Bound();
AssertEquals_LREAL(0.20657109030979783904, positionExtrema.Tmax, 1E-9, message:='Profile[0] Tmax incorrect');
AssertEquals_LREAL(-29.15176131633907630203, positionExtrema.Maximum, 1E-9, message:='Profile[0] maximum incorrect');
AssertEquals_LREAL(0.00000000000000000000, positionExtrema.Tmin, 1E-9, message:='Profile[0] Tmin incorrect');
AssertEquals_LREAL(-54.94342725690739825950, positionExtrema.Minimum, 1E-9, message:='Profile[0] minimum incorrect');

positionExtrema := ruckig._profiles[1].Bound();
AssertEquals_LREAL(0.19826331168683380968, positionExtrema.Tmax, 1E-9, message:='Profile[1] Tmax incorrect');
AssertEquals_LREAL(55.81702313192161568622, positionExtrema.Maximum, 1E-9, message:='Profile[1] maximum incorrect');
AssertEquals_LREAL(0.01113968648909354625, positionExtrema.Tmin, 1E-9, message:='Profile[1] Tmin incorrect');
AssertEquals_LREAL(-71.74511835894615785492, positionExtrema.Minimum, 1E-9, message:='Profile[1] minimum incorrect');

positionExtrema := ruckig._profiles[2].Bound();
AssertEquals_LREAL(0.22338925049474447904, positionExtrema.Tmax, 1E-9, message:='Profile[2] Tmax incorrect');
AssertEquals_LREAL(94.47974487226861128875, positionExtrema.Maximum, 1E-9, message:='Profile[2] maximum incorrect');
AssertEquals_LREAL(0.02606362117094545780, positionExtrema.Tmin, 1E-9, message:='Profile[2] Tmin incorrect');
AssertEquals_LREAL(-104.28684661857214166503, positionExtrema.Minimum, 1E-9, message:='Profile[2] minimum incorrect');
   

TEST_FINISHED();
END_METHOD

METHOD Test_Trajectory_HasTargetVelocity_HasTargetAcceleration_38
VAR_INST
  ruckig : Struckig.Otg(0.001, 3) := (
  
    Synchronization := SynchronizationType.TimeSync,        
    MaxVelocity := [ 2000.00000000000000000000, 2000.00000000000000000000, 2000.00000000000000000000 ],
    MaxAcceleration := [ 20000.00000000000000000000, 20000.00000000000000000000, 20000.00000000000000000000 ],
    MaxJerk := [ 800000.00000000000000000000, 800000.00000000000000000000, 800000.00000000000000000000 ],
    CurrentPosition := [ 70.18836201933098095651, -77.67370458831963730972, -11.76145133517785268396 ],
    CurrentVelocity := [ -105.04558581308560860634, 265.56449346599174532457, 964.37814674831179218017 ],
    CurrentAcceleration := [ -6039.95733145092708582524, -2777.20507650207400729414, 4352.81085492715828877408 ],
    TargetPosition := [ 71.40233970199534496714, 5.40303445887771260914, 92.98580498819549688960 ],
    TargetVelocity := [ -236.50355991826609169948, -66.98837676043160627160, 870.41763001953563616553 ],
    TargetAcceleration := [ -500.07275325607560034769, 72.93763981243137095589, -942.49209154303241575690 ]
  );
  
  positionExtrema : Struckig.ProfileBound;
END_VAR
TEST('Trajectory_HasTargetVelocity_HasTargetAcceleration_38');

ruckig();

// Check total duration of profiles
AssertEquals_LREAL(Expected := 0.14901888909886754075, Actual := ruckig.Duration, DELTA := 1E-8, Message := 'Duration incorrect');

// Check duration for each phase
positionExtrema := ruckig._profiles[0].Bound();
AssertEquals_LREAL(0.12406814159805865105, positionExtrema.Tmax, 1E-9, message:='Profile[0] Tmax incorrect');
AssertEquals_LREAL(75.12313380408009777511, positionExtrema.Maximum, 1E-9, message:='Profile[0] maximum incorrect');
AssertEquals_LREAL(0.02561480747291104351, positionExtrema.Tmin, 1E-9, message:='Profile[0] Tmin incorrect');
AssertEquals_LREAL(67.75537848504214366585, positionExtrema.Minimum, 1E-9, message:='Profile[0] minimum incorrect');

positionExtrema := ruckig._profiles[1].Bound();
AssertEquals_LREAL(0.13598633944686283614, positionExtrema.Tmax, 1E-9, message:='Profile[1] Tmax incorrect');
AssertEquals_LREAL(5.98711873384755755012, positionExtrema.Maximum, 1E-9, message:='Profile[1] maximum incorrect');
AssertEquals_LREAL(0.00000000000000000000, positionExtrema.Tmin, 1E-9, message:='Profile[1] Tmin incorrect');
AssertEquals_LREAL(-77.67370458831963730972, positionExtrema.Minimum, 1E-9, message:='Profile[1] minimum incorrect');

positionExtrema := ruckig._profiles[2].Bound();
AssertEquals_LREAL(0.14901888909886754075, positionExtrema.Tmax, 1E-9, message:='Profile[2] Tmax incorrect');
AssertEquals_LREAL(92.98580498819549688960, positionExtrema.Maximum, 1E-9, message:='Profile[2] maximum incorrect');
AssertEquals_LREAL(0.00000000000000000000, positionExtrema.Tmin, 1E-9, message:='Profile[2] Tmin incorrect');
AssertEquals_LREAL(-11.76145133517785268396, positionExtrema.Minimum, 1E-9, message:='Profile[2] minimum incorrect');
   

TEST_FINISHED();
END_METHOD

METHOD Test_Trajectory_HasTargetVelocity_HasTargetAcceleration_41
VAR_INST
  ruckig : Struckig.Otg(0.001, 3) := (
  
    Synchronization := SynchronizationType.TimeSync,        
    MaxVelocity := [ 2000.00000000000000000000, 2000.00000000000000000000, 2000.00000000000000000000 ],
    MaxAcceleration := [ 20000.00000000000000000000, 20000.00000000000000000000, 20000.00000000000000000000 ],
    MaxJerk := [ 800000.00000000000000000000, 800000.00000000000000000000, 800000.00000000000000000000 ],
    CurrentPosition := [ 77.70133891525995295524, 7.01592092562633240505, 41.88398938907070601090 ],
    CurrentVelocity := [ -954.47536643469038608600, -572.16261829852851406031, 473.16402135503631143365 ],
    CurrentAcceleration := [ -2847.17654342300011194311, -1889.61698757276462856680, -3110.21768918452016805531 ],
    TargetPosition := [ 92.37579717709354554245, -14.04614057772144519731, -73.88361356505039623244 ],
    TargetVelocity := [ 519.95772801058456025203, 127.89327712966064609645, -380.91422286825297760515 ],
    TargetAcceleration := [ -890.64075852453197512659, 681.51569675393488978443, 390.99828361762297390669 ]
  );
  
  positionExtrema : Struckig.ProfileBound;
END_VAR
TEST('Trajectory_HasTargetVelocity_HasTargetAcceleration_41');

ruckig();

// Check total duration of profiles
AssertEquals_LREAL(Expected := 0.18543052523247699481, Actual := ruckig.Duration, DELTA := 1E-8, Message := 'Duration incorrect');

// Check duration for each phase
positionExtrema := ruckig._profiles[0].Bound();
AssertEquals_LREAL(0.18543052523247699481, positionExtrema.Tmax, 1E-9, message:='Profile[0] Tmax incorrect');
AssertEquals_LREAL(92.37579717709354554245, positionExtrema.Maximum, 1E-9, message:='Profile[0] maximum incorrect');
AssertEquals_LREAL(0.07568410654937982041, positionExtrema.Tmin, 1E-9, message:='Profile[0] Tmin incorrect');
AssertEquals_LREAL(41.15768150995504015555, positionExtrema.Minimum, 1E-9, message:='Profile[0] minimum incorrect');

positionExtrema := ruckig._profiles[1].Bound();
AssertEquals_LREAL(0.00000000000000000000, positionExtrema.Tmax, 1E-9, message:='Profile[1] Tmax incorrect');
AssertEquals_LREAL(7.01592092562633240505, positionExtrema.Maximum, 1E-9, message:='Profile[1] maximum incorrect');
AssertEquals_LREAL(0.16752625845292970497, positionExtrema.Tmin, 1E-9, message:='Profile[1] Tmin incorrect');
AssertEquals_LREAL(-15.47801998831725711625, positionExtrema.Minimum, 1E-9, message:='Profile[1] minimum incorrect');

positionExtrema := ruckig._profiles[2].Bound();
AssertEquals_LREAL(0.02111222788851935261, positionExtrema.Tmax, 1E-9, message:='Profile[2] Tmax incorrect');
AssertEquals_LREAL(49.92568034606993876423, positionExtrema.Maximum, 1E-9, message:='Profile[2] maximum incorrect');
AssertEquals_LREAL(0.18543052523247699481, positionExtrema.Tmin, 1E-9, message:='Profile[2] Tmin incorrect');
AssertEquals_LREAL(-73.88361356505039623244, positionExtrema.Minimum, 1E-9, message:='Profile[2] minimum incorrect');
   

TEST_FINISHED();
END_METHOD

METHOD Test_Trajectory_HasTargetVelocity_HasTargetAcceleration_46
VAR_INST
  ruckig : Struckig.Otg(0.001, 3) := (
  
    Synchronization := SynchronizationType.TimeSync,        
    MaxVelocity := [ 2000.00000000000000000000, 2000.00000000000000000000, 2000.00000000000000000000 ],
    MaxAcceleration := [ 20000.00000000000000000000, 20000.00000000000000000000, 20000.00000000000000000000 ],
    MaxJerk := [ 800000.00000000000000000000, 800000.00000000000000000000, 800000.00000000000000000000 ],
    CurrentPosition := [ -81.70058267564624543411, -19.21897702137916041920, 94.53377990477645198553 ],
    CurrentVelocity := [ 791.96608977333426082623, 567.98007664216197554197, 949.19373974938935134560 ],
    CurrentAcceleration := [ -9852.41254141048739256803, -751.99368634466736693867, 3617.41551680202064744662 ],
    TargetPosition := [ 4.61526430014728816786, 47.19472748930556349478, -27.25527375543330776964 ],
    TargetVelocity := [ -365.39593288733976805815, -832.73312185042618693842, 15.48785727174674775597 ],
    TargetAcceleration := [ 393.54024330782590368472, -760.25458815149545444001, 23.06111995903222577908 ]
  );
  
  positionExtrema : Struckig.ProfileBound;
END_VAR
TEST('Trajectory_HasTargetVelocity_HasTargetAcceleration_46');

ruckig();

// Check total duration of profiles
AssertEquals_LREAL(Expected := 0.25941536116832880632, Actual := ruckig.Duration, DELTA := 1E-8, Message := 'Duration incorrect');

// Check duration for each phase
positionExtrema := ruckig._profiles[0].Bound();
AssertEquals_LREAL(0.23392343586419403478, positionExtrema.Tmax, 1E-9, message:='Profile[0] Tmax incorrect');
AssertEquals_LREAL(11.84902844379517183881, positionExtrema.Maximum, 1E-9, message:='Profile[0] maximum incorrect');
AssertEquals_LREAL(0.00000000000000000000, positionExtrema.Tmin, 1E-9, message:='Profile[0] Tmin incorrect');
AssertEquals_LREAL(-81.70058267564624543411, positionExtrema.Minimum, 1E-9, message:='Profile[0] minimum incorrect');

positionExtrema := ruckig._profiles[1].Bound();
AssertEquals_LREAL(0.19491405447314413824, positionExtrema.Tmax, 1E-9, message:='Profile[1] Tmax incorrect');
AssertEquals_LREAL(72.37093782213797510394, positionExtrema.Maximum, 1E-9, message:='Profile[1] maximum incorrect');
AssertEquals_LREAL(0.00000000000000000000, positionExtrema.Tmin, 1E-9, message:='Profile[1] Tmin incorrect');
AssertEquals_LREAL(-19.21897702137916041920, positionExtrema.Minimum, 1E-9, message:='Profile[1] minimum incorrect');

positionExtrema := ruckig._profiles[2].Bound();
AssertEquals_LREAL(0.02952176939600252917, positionExtrema.Tmax, 1E-9, message:='Profile[2] Tmax incorrect');
AssertEquals_LREAL(120.70144362619019773319, positionExtrema.Maximum, 1E-9, message:='Profile[2] maximum incorrect');
AssertEquals_LREAL(0.25322160979530433655, positionExtrema.Tmin, 1E-9, message:='Profile[2] Tmin incorrect');
AssertEquals_LREAL(-27.31907826634350300310, positionExtrema.Minimum, 1E-9, message:='Profile[2] minimum incorrect');
   

TEST_FINISHED();
END_METHOD

METHOD Test_Trajectory_HasTargetVelocity_HasTargetAcceleration_47
VAR_INST
  ruckig : Struckig.Otg(0.001, 3) := (
  
    Synchronization := SynchronizationType.TimeSync,        
    MaxVelocity := [ 2000.00000000000000000000, 2000.00000000000000000000, 2000.00000000000000000000 ],
    MaxAcceleration := [ 20000.00000000000000000000, 20000.00000000000000000000, 20000.00000000000000000000 ],
    MaxJerk := [ 800000.00000000000000000000, 800000.00000000000000000000, 800000.00000000000000000000 ],
    CurrentPosition := [ 81.61368863479273727535, 18.81647567172932156154, -89.15971183512543518646 ],
    CurrentVelocity := [ 614.05723536338791745948, 343.05287387529847364931, -371.00163086153361291508 ],
    CurrentAcceleration := [ 2762.36060607538092881441, -8252.84383845068077789620, 1522.48694311787949118298 ],
    TargetPosition := [ 31.53792392446635517445, -13.15393306556988761713, -67.81554985684867631335 ],
    TargetVelocity := [ 927.36256285251761255495, -453.39442766394324735302, -734.53754957298599492788 ],
    TargetAcceleration := [ -810.42747656261008160072, 683.82844872197824770410, -296.63416710646515639382 ]
  );
  
  positionExtrema : Struckig.ProfileBound;
END_VAR
TEST('Trajectory_HasTargetVelocity_HasTargetAcceleration_47');

ruckig();

// Check total duration of profiles
AssertEquals_LREAL(Expected := 0.25287606970423076591, Actual := ruckig.Duration, DELTA := 1E-8, Message := 'Duration incorrect');

// Check duration for each phase
positionExtrema := ruckig._profiles[0].Bound();
AssertEquals_LREAL(0.02845295075759422462, positionExtrema.Tmax, 1E-9, message:='Profile[0] Tmax incorrect');
AssertEquals_LREAL(97.13230269209392986340, positionExtrema.Maximum, 1E-9, message:='Profile[0] maximum incorrect');
AssertEquals_LREAL(0.22686303535852750390, positionExtrema.Tmin, 1E-9, message:='Profile[0] Tmin incorrect');
AssertEquals_LREAL(9.48720344289291794837, positionExtrema.Minimum, 1E-9, message:='Profile[0] minimum incorrect');

positionExtrema := ruckig._profiles[1].Bound();
AssertEquals_LREAL(0.02241468542399701822, positionExtrema.Tmax, 1E-9, message:='Profile[1] Tmax incorrect');
AssertEquals_LREAL(23.03639977720293785524, positionExtrema.Maximum, 1E-9, message:='Profile[1] maximum incorrect');
AssertEquals_LREAL(0.25287606970423076591, positionExtrema.Tmin, 1E-9, message:='Profile[1] Tmin incorrect');
AssertEquals_LREAL(-13.15393306556988761713, positionExtrema.Minimum, 1E-9, message:='Profile[1] minimum incorrect');

positionExtrema := ruckig._profiles[2].Bound();
AssertEquals_LREAL(0.20039624088411220337, positionExtrema.Tmax, 1E-9, message:='Profile[2] Tmax incorrect');
AssertEquals_LREAL(-46.06681198459425274905, positionExtrema.Maximum, 1E-9, message:='Profile[2] maximum incorrect');
AssertEquals_LREAL(0.03284040362274634473, positionExtrema.Tmin, 1E-9, message:='Profile[2] Tmin incorrect');
AssertEquals_LREAL(-95.92347928545005686374, positionExtrema.Minimum, 1E-9, message:='Profile[2] minimum incorrect');
   

TEST_FINISHED();
END_METHOD

METHOD Test_Trajectory_HasTargetVelocity_HasTargetAcceleration_48
VAR_INST
  ruckig : Struckig.Otg(0.001, 3) := (
  
    Synchronization := SynchronizationType.TimeSync,        
    MaxVelocity := [ 2000.00000000000000000000, 2000.00000000000000000000, 2000.00000000000000000000 ],
    MaxAcceleration := [ 20000.00000000000000000000, 20000.00000000000000000000, 20000.00000000000000000000 ],
    MaxJerk := [ 800000.00000000000000000000, 800000.00000000000000000000, 800000.00000000000000000000 ],
    CurrentPosition := [ -88.66208591478776668282, -31.58880789945652622919, 65.04291982806716987398 ],
    CurrentVelocity := [ 580.03497340359649570019, -746.36896556027750193607, 812.20588456619907447021 ],
    CurrentAcceleration := [ -6519.58462448879436124116, -9252.12079111587627266999, -5505.83185145304014440626 ],
    TargetPosition := [ -85.04127215306982634502, -92.28954144915404356198, -74.37698578032075147348 ],
    TargetVelocity := [ -365.82662455999411577068, -112.69189210154274860543, 154.77689249662125803297 ],
    TargetAcceleration := [ -682.87003825383567345852, -247.18670592987155032461, -122.60845320130738400621 ]
  );
  
  positionExtrema : Struckig.ProfileBound;
END_VAR
TEST('Trajectory_HasTargetVelocity_HasTargetAcceleration_48');

ruckig();

// Check total duration of profiles
AssertEquals_LREAL(Expected := 0.25037129752792702808, Actual := ruckig.Duration, DELTA := 1E-8, Message := 'Duration incorrect');

// Check duration for each phase
positionExtrema := ruckig._profiles[0].Bound();
AssertEquals_LREAL(0.04415928948418586242, positionExtrema.Tmax, 1E-9, message:='Profile[0] Tmax incorrect');
AssertEquals_LREAL(-76.79539758143890537667, positionExtrema.Maximum, 1E-9, message:='Profile[0] maximum incorrect');
AssertEquals_LREAL(0.00000000000000000000, positionExtrema.Tmin, 1E-9, message:='Profile[0] Tmin incorrect');
AssertEquals_LREAL(-88.66208591478776668282, positionExtrema.Minimum, 1E-9, message:='Profile[0] minimum incorrect');

positionExtrema := ruckig._profiles[1].Bound();
AssertEquals_LREAL(0.00000000000000000000, positionExtrema.Tmax, 1E-9, message:='Profile[1] Tmax incorrect');
AssertEquals_LREAL(-31.58880789945652622919, positionExtrema.Maximum, 1E-9, message:='Profile[1] maximum incorrect');
AssertEquals_LREAL(0.25037129752792697257, positionExtrema.Tmin, 1E-9, message:='Profile[1] Tmin incorrect');
AssertEquals_LREAL(-92.28954144915404356198, positionExtrema.Minimum, 1E-9, message:='Profile[1] minimum incorrect');

positionExtrema := ruckig._profiles[2].Bound();
AssertEquals_LREAL(0.01811771018568369973, positionExtrema.Tmax, 1E-9, message:='Profile[2] Tmax incorrect');
AssertEquals_LREAL(78.06162686897538094399, positionExtrema.Maximum, 1E-9, message:='Profile[2] maximum incorrect');
AssertEquals_LREAL(0.23054659268189173216, positionExtrema.Tmin, 1E-9, message:='Profile[2] Tmin incorrect');
AssertEquals_LREAL(-76.43062116116439597135, positionExtrema.Minimum, 1E-9, message:='Profile[2] minimum incorrect');
   

TEST_FINISHED();
END_METHOD

METHOD Test_Trajectory_HasTargetVelocity_HasTargetAcceleration_51
VAR_INST
  ruckig : Struckig.Otg(0.001, 3) := (
  
    Synchronization := SynchronizationType.TimeSync,        
    MaxVelocity := [ 2000.00000000000000000000, 2000.00000000000000000000, 2000.00000000000000000000 ],
    MaxAcceleration := [ 20000.00000000000000000000, 20000.00000000000000000000, 20000.00000000000000000000 ],
    MaxJerk := [ 800000.00000000000000000000, 800000.00000000000000000000, 800000.00000000000000000000 ],
    CurrentPosition := [ 52.80919631150752024951, -81.68038555889982887948, 42.06917442755320735159 ],
    CurrentVelocity := [ -848.38044536898496517097, -694.53443230755419790512, -67.27027959540748724976 ],
    CurrentAcceleration := [ -7839.42279939661148091545, 2086.65454098016925854608, -1769.91408787331420171540 ],
    TargetPosition := [ 18.36498902426966139956, 7.18108207234031681310, -24.86667965964299753523 ],
    TargetVelocity := [ -484.52530887106502177630, -330.54249305132475456048, 184.78707869201707580942 ],
    TargetAcceleration := [ 34.47472473095945133537, 524.15868234202798703336, 659.72269096659351816925 ]
  );
  
  positionExtrema : Struckig.ProfileBound;
END_VAR
TEST('Trajectory_HasTargetVelocity_HasTargetAcceleration_51');

ruckig();

// Check total duration of profiles
AssertEquals_LREAL(Expected := 0.22814955969060143892, Actual := ruckig.Duration, DELTA := 1E-8, Message := 'Duration incorrect');

// Check duration for each phase
positionExtrema := ruckig._profiles[0].Bound();
AssertEquals_LREAL(0.00000000000000000000, positionExtrema.Tmax, 1E-9, message:='Profile[0] Tmax incorrect');
AssertEquals_LREAL(52.80919631150752024951, positionExtrema.Maximum, 1E-9, message:='Profile[0] maximum incorrect');
AssertEquals_LREAL(0.06738171645932469755, positionExtrema.Tmin, 1E-9, message:='Profile[0] Tmin incorrect');
AssertEquals_LREAL(13.99608603958429142722, positionExtrema.Minimum, 1E-9, message:='Profile[0] minimum incorrect');

positionExtrema := ruckig._profiles[1].Bound();
AssertEquals_LREAL(0.20249436133767390045, positionExtrema.Tmax, 1E-9, message:='Profile[1] Tmax incorrect');
AssertEquals_LREAL(13.58224981559266097975, positionExtrema.Maximum, 1E-9, message:='Profile[1] maximum incorrect');
AssertEquals_LREAL(0.02239168182377478805, positionExtrema.Tmin, 1E-9, message:='Profile[1] Tmin incorrect');
AssertEquals_LREAL(-95.21214742443424938756, positionExtrema.Minimum, 1E-9, message:='Profile[1] minimum incorrect');

positionExtrema := ruckig._profiles[2].Bound();
AssertEquals_LREAL(0.00000000000000000000, positionExtrema.Tmax, 1E-9, message:='Profile[2] Tmax incorrect');
AssertEquals_LREAL(42.06917442755320735159, positionExtrema.Maximum, 1E-9, message:='Profile[2] maximum incorrect');
AssertEquals_LREAL(0.20746496504559683305, positionExtrema.Tmin, 1E-9, message:='Profile[2] Tmin incorrect');
AssertEquals_LREAL(-27.36779954300167716497, positionExtrema.Minimum, 1E-9, message:='Profile[2] minimum incorrect');
   

TEST_FINISHED();
END_METHOD

METHOD Test_Trajectory_HasTargetVelocity_HasTargetAcceleration_56
VAR_INST
  ruckig : Struckig.Otg(0.001, 3) := (
  
    Synchronization := SynchronizationType.TimeSync,        
    MaxVelocity := [ 2000.00000000000000000000, 2000.00000000000000000000, 2000.00000000000000000000 ],
    MaxAcceleration := [ 20000.00000000000000000000, 20000.00000000000000000000, 20000.00000000000000000000 ],
    MaxJerk := [ 800000.00000000000000000000, 800000.00000000000000000000, 800000.00000000000000000000 ],
    CurrentPosition := [ -75.10494070961726720270, -6.22395011546019816251, 35.64048680664691914899 ],
    CurrentVelocity := [ -825.41867748520257919154, -559.17669137031361970003, 331.05712850319173412572 ],
    CurrentAcceleration := [ -2748.49249899548522080295, -2734.78689775577458931366, 8828.96129221495357342064 ],
    TargetPosition := [ -88.93249178580995817356, 32.61549251092765189242, -4.33333209618611192582 ],
    TargetVelocity := [ -969.86803709259822880995, 219.52159207481986413768, 145.45315840784223837545 ],
    TargetAcceleration := [ 673.73439439858611876843, 589.54870253816602598818, 268.61037017006333371683 ]
  );
  
  positionExtrema : Struckig.ProfileBound;
END_VAR
TEST('Trajectory_HasTargetVelocity_HasTargetAcceleration_56');

ruckig();

// Check total duration of profiles
AssertEquals_LREAL(Expected := 0.22533279528439006945, Actual := ruckig.Duration, DELTA := 1E-8, Message := 'Duration incorrect');

// Check duration for each phase
positionExtrema := ruckig._profiles[0].Bound();
AssertEquals_LREAL(0.13546282954524005437, positionExtrema.Tmax, 1E-9, message:='Profile[0] Tmax incorrect');
AssertEquals_LREAL(-60.83093977470542768060, positionExtrema.Maximum, 1E-9, message:='Profile[0] maximum incorrect');
AssertEquals_LREAL(0.08546282954524006548, positionExtrema.Tmin, 1E-9, message:='Profile[0] Tmin incorrect');
AssertEquals_LREAL(-97.18448406099201974939, positionExtrema.Minimum, 1E-9, message:='Profile[0] minimum incorrect');

positionExtrema := ruckig._profiles[1].Bound();
AssertEquals_LREAL(0.22533279528439004169, positionExtrema.Tmax, 1E-9, message:='Profile[1] Tmax incorrect');
AssertEquals_LREAL(32.61549251092765189242, positionExtrema.Maximum, 1E-9, message:='Profile[1] maximum incorrect');
AssertEquals_LREAL(0.04813186201257521613, positionExtrema.Tmin, 1E-9, message:='Profile[1] Tmin incorrect');
AssertEquals_LREAL(-22.45997635018479243740, positionExtrema.Minimum, 1E-9, message:='Profile[1] minimum incorrect');

positionExtrema := ruckig._profiles[2].Bound();
AssertEquals_LREAL(0.04893648758049205100, positionExtrema.Tmax, 1E-9, message:='Profile[2] Tmax incorrect');
AssertEquals_LREAL(47.07359821757206930215, positionExtrema.Maximum, 1E-9, message:='Profile[2] maximum incorrect');
AssertEquals_LREAL(0.20659644161609555524, positionExtrema.Tmin, 1E-9, message:='Profile[2] Tmin incorrect');
AssertEquals_LREAL(-6.13445732070238047839, positionExtrema.Minimum, 1E-9, message:='Profile[2] minimum incorrect');
   

TEST_FINISHED();
END_METHOD

METHOD Test_Trajectory_HasTargetVelocity_HasTargetAcceleration_60
VAR_INST
  ruckig : Struckig.Otg(0.001, 3) := (
  
